(* CODESYS project twinsafe3diagnostics_v0.2.3.library
   Company: Beckhoff Automation LLC - Sample Code
   Version: 0.2.3
   Description: (Sample Code)
   Placeholder: TwinSafe3Diagnostics_v0.2.3
   Author: Jason Erickson
   Title: TwinSafe3Diagnostics_v0.2.3

Project tree, tasks and I/O mapping:
  libraries: Tc2_Drive, * (Beckhoff Automation GmbH); Tc2_EtherCAT, * (Beckhoff Automation GmbH); Tc2_MC2, * (Beckhoff Automation GmbH); Tc2_MC2_Drive, * (Beckhoff Automation GmbH); Tc2_Standard, * (Beckhoff Automation GmbH)
  DUTs/
    ConnectionAndFb_Data/
      FBs/
        data type ST_SAFETY_FB
      Project/
        data type ST_SAFETY_CONNECTION_AX5805
        data type ST_SAFETY_CONNECTION_EK1914
        data type ST_SAFETY_CONNECTION_EL1904
        data type ST_SAFETY_CONNECTION_EL2904
        data type ST_SAFETY_CONNECTION_EP1908
        data type ST_SAFETY_CONNECTION_GROUP
    HardwareData/
      data type ST_AX5805_DIAGNOSTICS
      data type ST_EK1914_DIAGNOSTICS
      data type ST_EL1904_DIAGNOSTICS
      data type ST_EL2904_DIAGNOSTICS
      data type ST_EL69xx_DIAGNOSTICS
      data type ST_EP1908_DIAGNOSTICS
  POUs/
    ConnectionAndFb_Blocks/
      FBs/
        function block FB_InfoAND [ST]
        function block FB_InfoConnectionShutdown [ST]
        function block FB_InfoDecoupler [ST]
        function block FB_InfoEDM [ST]
        function block FB_InfoEStop [ST]
        function block FB_InfoMON [ST]
        function block FB_InfoMuting [ST]
        function block FB_InfoOperationMode [ST]
        function block FB_InfoOR [ST]
        function block FB_InfoRS [ST]
        function block FB_InfoSR [ST]
        function block FB_InfoTOF [ST]
        function block FB_InfoTON [ST]
        function block FB_InfoTwoHand [ST]
      Project/
        function block FB_SafetyConnectionAX5805 [ST]
        function block FB_SafetyConnectionEK1914 [ST]
        function block FB_SafetyConnectionEL1904 [ST]
        function block FB_SafetyConnectionEL2904 [ST]
        function block FB_SafetyConnectionEP1908 [ST]
        function block FB_SafetyConnectionGroup [ST]
    HardwareFBs/
      function block FB_AX5805Diagnostics [ST]
      function block FB_EK1914Diagnostics [ST]
      function block FB_EL1904Diagnostics [ST]
      function block FB_EL2904Diagnostics [ST]
      function block FB_EL69xxDiagnostics [ST]
      function block FB_EP1908Diagnostics [ST]
  Version/
    global variables Global_Version
*)

// DUTs/ConnectionAndFb_Data/FBs/ST_SAFETY_FB
TYPE ST_SAFETY_FB :
STRUCT
(* ***** Structure variables individually linked to the 'Function Block Info Data' of the EL69xx. ***** *)
// State of the TwinSAFE FB.
	usiMapState: USINT;
// Diagnostics of the TwinSAFE FB.
	uiMapDiag: UINT;
END_STRUCT
END_TYPE

// DUTs/ConnectionAndFb_Data/Project/ST_SAFETY_CONNECTION_AX5805
TYPE ST_SAFETY_CONNECTION_AX5805 :
STRUCT
(* ***** Structure linked to the AX5805 'Connection Info Data' of the EL69xx. ***** *)
// State of the AX5805 TwinSAFE connection.
	usiMapState: USINT;
// Diagnostics of the AX5805 TwinSAFE connection.
	usiMapDiag: USINT;
// Connection Input Status signals of the AX5805.
	bInputSignals0: BYTE; // Input status of Channel 1 default motion functions and error.
	bInputSignals1: BYTE; // Input status of Channel 1 USER CONFIGURED motion functions and error.
	bInputSignals2: BYTE; // Input status of Channel 2 default motion functions and error.
	bInputSignals3: BYTE; // Input status of Channel 2 USER CONFIGURED motion functions and error.
// Connection Output Status signals of the AX5805.
	bOutputSignals0: BYTE; // Input status of Channel 1 default motion functions and error.
	bOutputSignals1: BYTE; // Input status of Channel 1 USER CONFIGURED motion functions and error.
	bOutputSignals2: BYTE; // Input status of Channel 2 default motion functions and error.
	bOutputSignals3: BYTE; // Input status of Channel 2 USER CONFIGURED motion functions and error.
END_STRUCT
END_TYPE

// DUTs/ConnectionAndFb_Data/Project/ST_SAFETY_CONNECTION_EK1914
TYPE ST_SAFETY_CONNECTION_EK1914 :
STRUCT
(* ***** Structure linked to the EK1914 'Connection Info Data' of the EL69xx. ***** *)
// State of the EK1914 TwinSAFE connection.
	usiMapState: USINT;
// Diagnostics of the EK1914 TwinSAFE connection.
	usiMapDiag: USINT;
// Input Safe Data Byte 0 of the EK1914.
	bInputSignals: BYTE;
// Output Safe Data Byte 0 of the EK1914.
	bOutputSignals: BYTE;
END_STRUCT
END_TYPE

// DUTs/ConnectionAndFb_Data/Project/ST_SAFETY_CONNECTION_EL1904
TYPE ST_SAFETY_CONNECTION_EL1904 :
STRUCT
(* ***** Structure linked to the EL1904 'Connection Info Data' of the EL69xx. ***** *)
// State of the EL1904 TwinSAFE connection.
	usiMapState: USINT;
// Diagnostics of the EL1904 TwinSAFE connection.
	usiMapDiag: USINT;
// Input Safe Data Byte 0 of the EL1904.
	bInputSignals: BYTE;
END_STRUCT
END_TYPE

// DUTs/ConnectionAndFb_Data/Project/ST_SAFETY_CONNECTION_EL2904
TYPE ST_SAFETY_CONNECTION_EL2904 :
STRUCT
(* ***** Structure linked to the EL2904 'Connection Info Data' of the EL69xx. ***** *)
// State of the EL2904 TwinSAFE connection.
	usiMapState: USINT;
// Diagnostics of the EL2904 TwinSAFE connection.
	usiMapDiag: USINT;
// Output Safe Data Byte 0 of the EL2904.
	bOutputSignals: BYTE;
END_STRUCT
END_TYPE

// DUTs/ConnectionAndFb_Data/Project/ST_SAFETY_CONNECTION_EP1908
TYPE ST_SAFETY_CONNECTION_EP1908 :
STRUCT
(* ***** Structure linked to the EP1908 'Connection Info Data' of the EL69xx. ***** *)
// State of the EP1908 TwinSAFE connection.
	usiMapState: USINT;
// Diagnostics of the EP1908 TwinSAFE connection.
	usiMapDiag: USINT;
// Input Safe Data Byte 0 of the EP1908.
	bInputSignals: BYTE;
END_STRUCT
END_TYPE

// DUTs/ConnectionAndFb_Data/Project/ST_SAFETY_CONNECTION_GROUP
TYPE ST_SAFETY_CONNECTION_GROUP :
STRUCT
(* ***** Structure linked to the 'TwinSAFE Group Info Data' of the EL69xx. ***** *)
// State of the EL2904 TwinSAFE Group.
	usiMapState: USINT;
// Diagnostics of the TwinSAFE Group.
	usiMapDiag: USINT;
END_STRUCT
END_TYPE

// DUTs/HardwareData/ST_AX5805_DIAGNOSTICS
TYPE ST_AX5805_DIAGNOSTICS :
STRUCT
// Serial number of the AX5805.
	dwSerialNumber: DWORD;
// DIP Switch setting of the AX5805.
	wDipSwitch: WORD;
// Hardware Version of the AX5805.
	sHwVersion: STRING(2);
// Software/Firmware Version of the AX5805.
	sFwVersion: STRING(2);
// Micro Controller (MC1) Temperature in DegC of the AX5805.
	wMC1Temp: WORD;
	xMC1_TempHighAlarm: BOOL;
	xMC1_TempLowAlarm: BOOL;
// Micro Controller (MC2) Temperature in DegC of the AX5805.
	wMC2Temp: WORD;
	xMC2_TempHighAlarm: BOOL;
	xMC2_TempLowAlarm: BOOL;
// Micro Controller (MC1) Voltage in mV of the AX5805.
	lrMC1_3300mV: LREAL;
	lrMC1_5000mV: LREAL;
	xMC1_SupplyVoltHighAlarm: BOOL;
	xMC1_SupplyVoltLowAlarm: BOOL;
// Micro Controller (MC2) Voltage (mV) of the AX5805.
	lrMC2_3300mV: LREAL;
	lrMC2_5000mV: LREAL;
	xMC2_SupplyVoltHighAlarm: BOOL;
	xMC2_SupplyVoltLowAlarm: BOOL;
// Configured Safety Option of the AX5000 Drive.
	sSafetyOption: STRING(25);
// Diagnostics outputs of the AX5805.
	sDiagReason: STRING(255);
	sDiagReaction: STRING;
	xDiagnosticAlarm: BOOL;
	iDiagIndex: INT;
// Error outputs of the AX5805.
	sErrorName: STRING;
	sErrorDescription: STRING(255);
	xErrorAlarm: BOOL;
	iErrorIndex: INT;
// Connection State of the AX5805.
	sConnectionState: STRING;
// Error Status of the AX5805.
	xAX5805Error: BOOL;
END_STRUCT
END_TYPE

// DUTs/HardwareData/ST_EK1914_DIAGNOSTICS
TYPE ST_EK1914_DIAGNOSTICS :
STRUCT
// Serial number of the EK1914.
	dwSerialNumber: DWORD;
// DIP Switch setting of the EK1914.
	wDipSwitch: WORD;
// Hardware version of the EK1914.
	sHwVersion: STRING;
// Software/Firmware version of the EK1914.
	sFwVersion: STRING;
// Micro Controller Temperature in DegC of the EK1914.
	wMC1Temp: WORD;
	wMC2Temp: WORD;
// Micro Controller Voltage in mV of the EK1914.
	lrMC1_3300mV: LREAL;
	lrMC2_3300mV: LREAL;
// Sensor Tests Active of the EK1914.
	xSensorTestActive1: BOOL;
	xSensorTestActive2: BOOL;
// Sensor Test Errors of the EK1914.
	xSensorTest1_Error: BOOL;
	xSensorTest2_Error: BOOL;
// Logic Mode of the EK1914 Channels 1 & 2.
	sLogicMode_Ch1Ch2: STRING;
// Standard Output Active/Inactive of the EK1914.
	xStandardOutputActive: BOOL;	
//Test Pulses Active/Inactive of the EK1914.
	xTestPulsesActive: BOOL;
//Output Error Acknowledge Active/Inactive of the EK1914.
	xOutputErrAckActive: BOOL;
// Two-Channel Evaluation Error of the EK1914.
	x2ChanEvalError_Pair1: BOOL;
// Safety Mat Mode Error of the EK1914.
	xSafeMatError_Pair1: BOOL;
// Safety Mat External Supply error of the EK1914.
	xSafeMatExternalSupplyErrorCh1: BOOL;
	xSafeMatExternalSupplyErrorCh2: BOOL;
// Error At The Output of the EK1914 (MC1).
	sOutputErrorDescription_MC1: STRING;
	xCrossCircuitError1_MC1: BOOL;
	xCrossCircuitError2_MC1: BOOL;
	xOverVoltage_MC1: BOOL;
	xUnderVoltage_MC1: BOOL;
	xFieldVoltageError_MC1: BOOL;
	xStartupOutCircuitError_MC1: BOOL;
	xExternalSupply0vError1_MC1: BOOL;
	xExternalSupply24vError1_MC1: BOOL;
	xExternalSupply0vError2_MC1: BOOL;
	xExternalSupply24vError2_MC1: BOOL;
// Error At The Output of the EK1914 (MC2).
	sOutputErrorDescription_MC2: STRING;
	xCrossCircuitError1_MC2: BOOL;
	xCrossCircuitError2_MC2: BOOL;
	xOverVoltage_MC2: BOOL;
	xUnderVoltage_MC2: BOOL;
	xFieldVoltageError_MC2: BOOL;
	xStartupOutCircuitError_MC2: BOOL;
	xExternalSupply0vError1_MC2: BOOL;
	xExternalSupply24vError1_MC2: BOOL;
	xExternalSupply0vError2_MC2: BOOL;
	xExternalSupply24vError2_MC2: BOOL;
// Connection State of the EK1914.
	sConnectionState: STRING;
// Error Status of the EK1914.
	xEK1914Error: BOOL;
END_STRUCT
END_TYPE

// DUTs/HardwareData/ST_EL1904_DIAGNOSTICS
TYPE ST_EL1904_DIAGNOSTICS :
STRUCT
// Serial number of the EL1904.
	dwSerialNumber: DWORD;
// DIP Switch setting of the EL1904.
	wDipSwitch: WORD;
// Hardware version of the EL1904.
	sHwVersion: STRING;
// Software/Firmware version of the EL1904.
	sFwVersion: STRING;
// Micro Controller Temperature in DegC of the EL1904.
	wMC1Temp: WORD;
	wMC2Temp: WORD;
// Micro Controller Voltage in mV of the EL1904.
	lrMC1_3300mV: LREAL;
	lrMC2_3300mV: LREAL;
// Operating Mode of the EL1904.
	sOpMode: STRING;
// Sensor Tests Active of the EL1904.
	xSensorTestActive1: BOOL;
	xSensorTestActive2: BOOL;
	xSensorTestActive3: BOOL;
	xSensorTestActive4: BOOL;
// Sensor Test Errors of the EL1904.
	xSensorTest1_Error: BOOL;
	xSensorTest2_Error: BOOL;
	xSensorTest3_Error: BOOL;
	xSensorTest4_Error: BOOL;
// Logic Mode of the EL1904 Channels 1 & 2.
	sLogicMode_Ch1Ch2: STRING;
// Logic Mode of the EL1904 Channels 3 & 4.
	sLogicMode_Ch3Ch4: STRING;
// Two-Channel Evaluation Error of the EL1904.
	x2ChanEvalError_Pair1: BOOL;
	x2ChanEvalError_Pair2: BOOL;
// Safety Mat Mode Error of the EL1904.
	xSafeMatError_Pair1: BOOL;
	xSafeMatError_Pair2: BOOL;
// Safety Mat External Supply error of the EL1904.
	xSafeMatExternalSupplyErrorCh1: BOOL;
	xSafeMatExternalSupplyErrorCh2: BOOL;
	xSafeMatExternalSupplyErrorCh3: BOOL;
	xSafeMatExternalSupplyErrorCh4: BOOL;
// Connection State of the EL1904.
	sConnectionState: STRING;
// Error Status of the EL1904.
	xEL1904Error: BOOL;
END_STRUCT
END_TYPE

// DUTs/HardwareData/ST_EL2904_DIAGNOSTICS
TYPE ST_EL2904_DIAGNOSTICS :
STRUCT
// Serial number of the EL2904.
	dwSerialNumber: DWORD;
// DIP Switch setting of the EL2904.
	wDipSwitch: WORD;
// Hardware version of the EL2904.
	sHwVersion: STRING;
// Software/Firmware version of the EL2904.
	sFwVersion: STRING;
// Micro Controller Temperature in DegC of the EL2904.
	wMC1Temp: WORD;
	wMC2Temp: WORD;
// Micro Controller Voltage in mV of the EL2904.
	lrMC1_3300mV: LREAL;
	lrMC2_3300mV: LREAL;
// Standard Output Active/Inactive of the EL2904.
	xStandardOutputActive: BOOL;	
// Current Measurement Active of the EL2904.
	xCurrentMeasureActive: BOOL;
//Test Pulses Active/Inactive of the EL2904.
	xTestPulsesActive: BOOL;
//Output Error Acknowledge Active/Inactive of the EL2904.
	xOutputErrAckActive: BOOL;
// Error At The Output of the EL2904.
	xExternalSupplyOrCrossCircuitError1: BOOL;
	xExternalSupplyOrCrossCircuitError2: BOOL;
	xExternalSupplyOrCrossCircuitError3: BOOL;
	xExternalSupplyOrCrossCircuitError4: BOOL;
	xLoadError1: BOOL;
	xLoadError2: BOOL;
	xLoadError3: BOOL;
	xLoadError4: BOOL;
//Power Rail Supply Error of the EL2904
	xPowerRailSupplyVoltHighError: BOOL;
	xPowerRailSupplyVoltLowError: BOOL;
// Internal Chip Temperature Error of the EL2904.
	xOverTempMC1: BOOL;
	xOverTempMC2: BOOL;
	xOverTempOutputBoard: BOOL;
	xUnderTempMC1: BOOL;
	xUnderTempMC2: BOOL;
	xUnderTempOutputBoard: BOOL;
	xTempDiffOutputBoard: BOOL;
	xTempDiff_MC1MC2: BOOL;
// Connection State of the EL2904.
	sConnectionState: STRING;
// Error Status of the EL2904.
	xEL2904Error: BOOL;
END_STRUCT
END_TYPE

// DUTs/HardwareData/ST_EL69xx_DIAGNOSTICS
TYPE ST_EL69xx_DIAGNOSTICS :
STRUCT
// Serial number of the EL69xx.
	dwSerialNumber: DWORD;
// DIP Switch setting of the EL69xx.
	wDipSwitch: WORD;
// Hardware version of the EL69xx.
	sHwVersion: STRING;
// Software/Firmware version of the EL69xx.
	sFwVersion: STRING;
// Micro Controller Temperature in DegC of the EL69xx.
	wMC1Temp: WORD;
	wMC2Temp: WORD;
// Micro Controller voltage in mV of the EL69xx.
	lrMC1_3300mV: LREAL;
	lrMC2_3300mV: LREAL;
// Temperature and Voltage Errors of the EL69xx.
	xMaxTempError: BOOL;
	xMinTempError: BOOL;
	xTempDiffError: BOOL;
	xMaxVccMC1: BOOL;
	xMaxVccMC2: BOOL;
	xMinVccMC1: BOOL;
	xMinVccMC2: BOOL;
// Number Of Connections Configured in the EL69xx.
	bNumOfConnections: BYTE;
// Number of Safety Groups Configured in the EL69xx.
	bNumOfSafetyGroups: BYTE;
//Number of Safety Function Blocks Configured in the EL69xx.
	bNumOfSafetyBlocks: BYTE;
// Error Status of the EL69xx.
	xEL69xxError: BOOL;
END_STRUCT
END_TYPE

// DUTs/HardwareData/ST_EP1908_DIAGNOSTICS
TYPE ST_EP1908_DIAGNOSTICS :
STRUCT
// Serial number of the EP1908.
	dwSerialNumber: DWORD;
// DIP Switch setting of the EP1908.
	wDipSwitch: WORD;
// Hardware version of the EP1908.
	sHwVersion: STRING;
// Software/Firmware version of the EP1908.
	sFwVersion: STRING;
// Micro Controller Temperature in DegC of the EP1908.
	wMC1Temp: WORD;
	wMC2Temp: WORD;
// Micro Controller Voltage in mV of the EP1908.
	lrMC1_3300mV: LREAL;
	lrMC2_3300mV: LREAL;
// Operating Mode of the EP1908.
	sOpMode: STRING;
// Sensor Tests Active of the EP1908.
	xSensorTestActive1: BOOL;
	xSensorTestActive2: BOOL;
	xSensorTestActive3: BOOL;
	xSensorTestActive4: BOOL;
	xSensorTestActive5: BOOL;
	xSensorTestActive6: BOOL;
	xSensorTestActive7: BOOL;
	xSensorTestActive8: BOOL;
// Sensor Test Errors of the EP1908.
	xSensorTest1_Error: BOOL;
	xSensorTest2_Error: BOOL;
	xSensorTest3_Error: BOOL;
	xSensorTest4_Error: BOOL;
	xSensorTest5_Error: BOOL;
	xSensorTest6_Error: BOOL;
	xSensorTest7_Error: BOOL;
	xSensorTest8_Error: BOOL;
// Logic Mode 1 & 2 of the EP1908.
	sLogicMode_Ch1Ch2: STRING;
// Logic Mode 3 & 4 of the EP1908.
	sLogicMode_Ch3Ch4: STRING;
// Logic Mode 5 & 6 of the EP1908.
	sLogicMode_Ch5Ch6: STRING;
// Logic Mode 7 & 8 of the EP1908.
	sLogicMode_Ch7Ch8: STRING;
// Velocity/Frequency Limits of the EP1908.
	iEP1908_VelocityLimitCh1: INT;
	iEP1908_VelocityLimitCh2: INT;
	iEP1908_VelocityLimitCh3: INT;
	iEP1908_VelocityLimitCh4: INT;
	iEP1908_VelocityLimitCh5: INT;
	iEP1908_VelocityLimitCh6: INT;
	iEP1908_VelocityLimitCh7: INT;
	iEP1908_VelocityLimitCh8: INT;
// Actual Velocity/Frequencies of the EP1908.
 	iEP1908_ActVeloctiyCh1: INT;
 	iEP1908_ActVeloctiyCh2: INT;
 	iEP1908_ActVeloctiyCh3: INT;
 	iEP1908_ActVeloctiyCh4: INT;
 	iEP1908_ActVeloctiyCh5: INT;
 	iEP1908_ActVeloctiyCh6: INT;
 	iEP1908_ActVeloctiyCh7: INT;
 	iEP1908_ActVeloctiyCh8: INT;
// Max Velocitys/Frequencies of the EP1908.
	iEP1908_MaxVeloctiyCh1: INT;
	iEP1908_MaxVeloctiyCh2: INT;
	iEP1908_MaxVeloctiyCh3: INT;
	iEP1908_MaxVeloctiyCh4: INT;
	iEP1908_MaxVeloctiyCh5: INT;
	iEP1908_MaxVeloctiyCh6: INT;
	iEP1908_MaxVeloctiyCh7: INT;
	iEP1908_MaxVeloctiyCh8: INT;
// Two-Channel Evaluation Error of the EP1908.
	x2ChanEvalError_Pair1: BOOL;
	x2ChanEvalError_Pair2: BOOL;
	x2ChanEvalError_Pair3: BOOL;
	x2ChanEvalError_Pair4: BOOL;
// Safety Mat Mode Error of the EP1908.
	xSafeMatError_Pair1: BOOL;
	xSafeMatError_Pair2: BOOL;
	xSafeMatError_Pair3: BOOL;
	xSafeMatError_Pair4: BOOL;
// Safety Mat External Supply error of the EP1908.
	xSafeMatExternalSupplyErrorCh1: BOOL;
	xSafeMatExternalSupplyErrorCh2: BOOL;
	xSafeMatExternalSupplyErrorCh3: BOOL;
	xSafeMatExternalSupplyErrorCh4: BOOL;
	xSafeMatExternalSupplyErrorCh5: BOOL;
	xSafeMatExternalSupplyErrorCh6: BOOL;
	xSafeMatExternalSupplyErrorCh7: BOOL;
	xSafeMatExternalSupplyErrorCh8: BOOL;
// Speed Monitoring Error: Overspeed of the EP1908. 
// (Overspeed was detected at the input).
	xSpeedMonitorErrorCh1: BOOL;
	xSpeedMonitorErrorCh2: BOOL;
	xSpeedMonitorErrorCh3: BOOL;
	xSpeedMonitorErrorCh4: BOOL;
	xSpeedMonitorErrorCh5: BOOL;
	xSpeedMonitorErrorCh6: BOOL;
	xSpeedMonitorErrorCh7: BOOL;
	xSpeedMonitorErrorCh8: BOOL;
// Two Channel Sync Velocity Control Error of the EP1908. 
// (Both inputs of an input pair were read with inactive State).
	x2ChSyncVelocityErrorPair1: BOOL;
	x2ChSyncVelocityErrorPair2: BOOL;
	x2ChSyncVelocityErrorPair3: BOOL;
	x2ChSyncVelocityErrorPair4: BOOL;
// Two Channel Sync Velocity AND Two Channel Encoder Velocity Error of the EP1908.
// (Different speeds were identified for the two inputs of an input pair).
	x2ChSyncVeloAnd2ChEncVeloErrorPair1: BOOL;
	x2ChSyncVeloAnd2ChEncVeloErrorPair2: BOOL;
	x2ChSyncVeloAnd2ChEncVeloErrorPair3: BOOL;
	x2ChSyncVeloAnd2ChEncVeloErrorPair4: BOOL;
// Connection State of the EP1908.
	sConnectionState: STRING;
// Error Status of the EP1908.
	xEP1908Error: BOOL;
END_STRUCT
END_TYPE

// Version/Global_Version
// This function has been automatically generated from the project information.
VAR_GLOBAL CONSTANT
	{attribute 'const_non_replaced'}
	{attribute 'linkalways'}
	stLibVersion_TwinSafe3Diagnostics_v0_2_3 : ST_LibVersion := (iMajor := 0, iMinor := 2, iBuild := 3, iRevision := 0, sVersion := '0.2.3');
END_VAR

// POUs/ConnectionAndFb_Blocks/FBs/FB_InfoAND
(*=====================================================================
Beckhoff Automation LLC
Copyright 2015 All Rights Reserved
=======================================================================
Description: 
This Program has been supplied by Beckhoff Automation As-Is and is intended only as an example implementation. 
Functionality is not guaranteed. 
This Function Block reads status and error information known at time of creation of the TwinSAFE 'safeAnd' 
function block.
---------------------------------------------------------------------------------------------------------------
History:
Date		Version			Author							Comment
---------------------------------------------------------------------------------------------------------------
07.08.15	0.10		Jason Erickson				Initial Library Creation.
07.20.15	0.11		Jason Ericskon				Added CoE Read for TwinSAFE Connection State.
08.28.15	0.20		Jason Erickson				Code optimization to eliminate timed data reads.
09.18.15	0.2.1		Jason Erickson				Added new error codes 0x6000 - 0x6002 and Connection Status
														to the AX5805.
*)
FUNCTION_BLOCK FB_InfoAND
VAR_INPUT
(* ***** Structure variables individually linked to the 'Function Block Info Data' of the EL69xx. ***** *)
	i_stInfoData: ST_SAFETY_FB ;
END_VAR
VAR_OUTPUT
// State of the TwinSAFE FB.
	q_sState: STRING ;
END_VAR

// Evaluate safeAnd FB State.
IF i_stInfoData.usiMapState = 0 THEN
	q_sState := 'Undefined' ;
	ELSIF i_stInfoData.usiMapState 	= 	1 THEN
		q_sState := 'RUN' ;
	ELSIF i_stInfoData.usiMapState = 2 THEN
		q_sState := 'STOP' ;
	ELSIF i_stInfoData.usiMapState = 3 THEN
		q_sState := 'SAFE' ;
	ELSE
		q_sState := 'Unknown' ;
END_IF

// THE 'safeAnd' FB HAS NO DIAGNISTIC BYTE TO DECODE!

END_FUNCTION_BLOCK

// POUs/ConnectionAndFb_Blocks/FBs/FB_InfoConnectionShutdown
(*=====================================================================
Beckhoff Automation LLC
Copyright 2015 All Rights Reserved
=======================================================================
Description: 
This Program has been supplied by Beckhoff Automation As-Is and is intended only as an example implementation. 
Functionality is not guaranteed. 
This Function Block reads status and error information known at time of creation of the TwinSAFE 'safeConnShutdown' 
function block.
---------------------------------------------------------------------------------------------------------------
History:
Date		Version			Author							Comment
---------------------------------------------------------------------------------------------------------------
07.08.15	0.10		Jason Erickson				Initial Library Creation.
07.20.15	0.11		Jason Ericskon				Added CoE Read for TwinSAFE Connection State.
08.28.15	0.20		Jason Erickson				Code optimization to eliminate timed data reads.
09.18.15	0.2.1		Jason Erickson				Added new error codes 0x6000 - 0x6002 and Connection Status
														to the AX5805.
*)
FUNCTION_BLOCK FB_InfoConnectionShutdown
VAR_INPUT
(* ***** Structure variables individually linked to the 'Function Block Info Data' of the EL69xx. ***** *)
	i_stInfoData: ST_SAFETY_FB ;
END_VAR
VAR_OUTPUT
// State of the TwinSAFE FB.
	q_sState: STRING ;
// Diagnostics of the TwinSAFE FB.
	q_sDiag: STRING ;
END_VAR

// Evaluate safeConnShutdown FB State.
IF i_stInfoData.usiMapState = 0 THEN
	q_sState := 'Undefined' ;
	ELSIF i_stInfoData.usiMapState = 2 THEN
		q_sState := 'STOP' ;
	ELSIF i_stInfoData.usiMapState 	= 	3 THEN
		q_sState := 'SAFE' ;
	ELSIF i_stInfoData.usiMapState = 4 THEN
		q_sState := 'Error' ;
	ELSIF i_stInfoData.usiMapState = 5 THEN
		q_sState := 'Reset' ;
	ELSIF i_stInfoData.usiMapState = 10 THEN
		q_sState := 'Active' ;
	ELSIF i_stInfoData.usiMapState = 11 THEN
		q_sState := 'Deactive' ;
	ELSE
		q_sState := 'Unknown' ;
END_IF

// Evaluate safeConnShutdown FB Diagnostics.
IF i_stInfoData.uiMapDiag = 0 THEN
	q_sDiag := 'No Error' ;
	ELSIF  i_stInfoData.uiMapDiag = 1 THEN
		q_sDiag := 'Discrepancy Error Input Group1' ;
	ELSE
		q_sDiag := 'Unknown' ;
END_IF

END_FUNCTION_BLOCK

// POUs/ConnectionAndFb_Blocks/FBs/FB_InfoDecoupler
(*=====================================================================
Beckhoff Automation LLC
Copyright 2015 All Rights Reserved
=======================================================================
Description: 
This Program has been supplied by Beckhoff Automation As-Is and is intended only as an example implementation. 
Functionality is not guaranteed. 
This Function Block reads status and error information known at time of creation of the TwinSAFE 'safeDecouple' 
function block.
---------------------------------------------------------------------------------------------------------------
History:
Date		Version			Author							Comment
---------------------------------------------------------------------------------------------------------------
07.08.15	0.10		Jason Erickson				Initial Library Creation.
07.20.15	0.11		Jason Ericskon				Added CoE Read for TwinSAFE Connection State.
08.28.15	0.20		Jason Erickson				Code optimization to eliminate timed data reads.
09.18.15	0.2.1		Jason Erickson				Added new error codes 0x6000 - 0x6002 and Connection Status
														to the AX5805.
*)
FUNCTION_BLOCK FB_InfoDecoupler
VAR_INPUT
(* ***** Structure variables individually linked to the 'Function Block Info Data' of the EL69xx. ***** *)
	i_stInfoData: ST_SAFETY_FB ;
END_VAR
VAR_OUTPUT
// State of the TwinSAFE FB.
	q_sState: STRING ;
END_VAR

// Evaluate safeDecouple FB State.
IF i_stInfoData.usiMapState = 0 THEN
	q_sState := 'Undefined' ;
	ELSIF i_stInfoData.usiMapState = 1 THEN
		q_sState := 'RUN' ;
	ELSIF i_stInfoData.usiMapState = 2 THEN
		q_sState := 'STOP' ;
	ELSE
		q_sState := 'Unknown' ;
END_IF

// THE 'DECOUPLE FB' HAS NO DIAGNOSTIC BYTE TO DECODE!

END_FUNCTION_BLOCK

// POUs/ConnectionAndFb_Blocks/FBs/FB_InfoEDM
(*=====================================================================
Beckhoff Automation LLC
Copyright 2015 All Rights Reserved
=======================================================================
Description: 
This Program has been supplied by Beckhoff Automation As-Is and is intended only as an example implementation. 
Functionality is not guaranteed. 
This Function Block reads status and error information known at time of creation of the TwinSAFE 'safeEdm' 
function block.
---------------------------------------------------------------------------------------------------------------
History:
Date		Version			Author							Comment
---------------------------------------------------------------------------------------------------------------
07.08.15	0.10		Jason Erickson				Initial Library Creation.
07.20.15	0.11		Jason Ericskon				Added CoE Read for TwinSAFE Connection State.
08.28.15	0.20		Jason Erickson				Code optimization to eliminate timed data reads.
09.18.15	0.2.1		Jason Erickson				Added new error codes 0x6000 - 0x6002 and Connection Status
														to the AX5805.
*)
FUNCTION_BLOCK FB_InfoEDM
VAR_INPUT
(* ***** Structure variables individually linked to the 'Function Block Info Data' of the EL69xx. ***** *)
	i_stInfoData: ST_SAFETY_FB ;
END_VAR
VAR_OUTPUT
// State of the TwinSAFE FB.
	q_sState: STRING ;
// Diagnostics of the TwinSAFE FB.
	q_sDiag: STRING ;
END_VAR

// Evaluate safeEdm FB State.
IF i_stInfoData.usiMapState = 0 THEN
				q_sState := 'Undefined' ;
	ELSIF i_stInfoData.usiMapState = 2 THEN
				q_sState := 'STOP' ;
	ELSIF i_stInfoData.usiMapState = 4 THEN
				q_sState := 'ERROR' ;
	ELSIF i_stInfoData.usiMapState 	= 	5 THEN
				q_sState := 'RESET' ;
	ELSIF i_stInfoData.usiMapState = 14 THEN
				q_sState := 'Monitor-OFF' ;
	ELSIF i_stInfoData.usiMapState = 15 THEN
				q_sState := 'Monitor-ON' ;
	ELSE
				q_sState := 'Unknown' ;
END_IF

// Evaluate safeEdm FB Diagnostics
IF i_stInfoData.uiMapDiag = 0 THEN
				q_sDiag := 'No Error' ;
ELSIF  i_stInfoData.uiMapDiag = 1 THEN
				q_sDiag	:= 'Switch-OFF Timer Elapsed' ;
ELSIF  i_stInfoData.uiMapDiag = 2 THEN
				q_sDiag := 'Switch-ON Timer Elapsed' ;
ELSE
				q_sDiag := 'Unknown' ;
END_IF

END_FUNCTION_BLOCK

// POUs/ConnectionAndFb_Blocks/FBs/FB_InfoEStop
(*=====================================================================
Beckhoff Automation LLC
Copyright 2015 All Rights Reserved
=======================================================================
Description: 
This Program has been supplied by Beckhoff Automation As-Is and is intended only as an example implementation. 
Functionality is not guaranteed. 
This Function Block reads status and error information known at time of creation of the TwinSAFE 'safeEstop' 
function block.
---------------------------------------------------------------------------------------------------------------
History:
Date		Version			Author							Comment
---------------------------------------------------------------------------------------------------------------
07.08.15	0.10		Jason Erickson				Initial Library Creation.
07.20.15	0.11		Jason Ericskon				Added CoE Read for TwinSAFE Connection State.
08.28.15	0.20		Jason Erickson				Code optimization to eliminate timed data reads.
09.18.15	0.2.1		Jason Erickson				Added new error codes 0x6000 - 0x6002 and Connection Status
														to the AX5805.
*)
FUNCTION_BLOCK FB_InfoEStop
VAR_INPUT
(* ***** Structure variables individually linked to the 'Function Block Info Data' of the EL69xx. ***** *)
	i_stInfoData: ST_SAFETY_FB ;
END_VAR
VAR_OUTPUT
// State of the TwinSAFE FB.
	q_sState: STRING ;
// Diagnostics of the TwinSAFE FB.
	q_sDiag: STRING ;
END_VAR

// Evaluate state of the TwinSAFE 'ESTOP' FB.
IF i_stInfoData.usiMapState = 0 THEN
	q_sState := 'Undefined' ;
	ELSIF i_stInfoData.usiMapState = 1 THEN
		q_sState := 'RUN' ;
	ELSIF i_stInfoData.usiMapState = 2 THEN
		q_sState := 'STOP' ;
	ELSIF i_stInfoData.usiMapState = 3 THEN
		q_sState := 'SAFE' ;
	ELSIF i_stInfoData.usiMapState = 4 THEN
		q_sState := 'ERROR' ;
	ELSIF i_stInfoData.usiMapState = 5 THEN
		q_sState := 'RESET' ;
	ELSIF i_stInfoData.usiMapState = 6 THEN
		q_sState := 'START' ;
	ELSIF i_stInfoData.usiMapState = 8 THEN
		q_sState := 'DELAYOUT' ;
	ELSE
		q_sState := 'Unknown' ;
END_IF

// Evaluate diagnostics of the TwinSAFE 'ESTOP' FB.
IF i_stInfoData.uiMapDiag = 0 THEN
	q_sDiag := 'No Error' ;
	ELSIF i_stInfoData.uiMapDiag = 1 THEN
		q_sDiag := 'Discrepancy Error Input Group 1' ;
	ELSIF i_stInfoData.uiMapDiag = 2 THEN
		q_sDiag := 'Discrepancy Error Input Group 2' ;
	ELSIF i_stInfoData.uiMapDiag = 4 THEN
		q_sDiag := 'Discrepancy Error Input Group 3' ;
	ELSIF i_stInfoData.uiMapDiag = 8 THEN
		q_sDiag := 'Discrepancy Error Input Group 4' ;
	ELSIF i_stInfoData.uiMapDiag = 16 THEN
		q_sDiag := 'EDM 1 Monitoring Error' ;	
	ELSIF i_stInfoData.uiMapDiag = 32 THEN
		q_sDiag :=  	'EDM 2 Monitoring Error' ;	
	ELSE
		q_sDiag := 'Unknown' ;
END_IF

END_FUNCTION_BLOCK

// POUs/ConnectionAndFb_Blocks/FBs/FB_InfoMON
(*=====================================================================
Beckhoff Automation LLC
Copyright 2015 All Rights Reserved
=======================================================================
Description: 
This Program has been supplied by Beckhoff Automation As-Is and is intended only as an example implementation. 
Functionality is not guaranteed. 
This Function Block reads status and error information known at time of creation of the TwinSAFE 'safeMon' 
function block.
---------------------------------------------------------------------------------------------------------------
History:
Date		Version			Author							Comment
---------------------------------------------------------------------------------------------------------------
07.08.15	0.10		Jason Erickson				Initial Library Creation.
07.20.15	0.11		Jason Ericskon				Added CoE Read for TwinSAFE Connection State.
08.28.15	0.20		Jason Erickson				Code optimization to eliminate timed data reads.
09.18.15	0.2.1		Jason Erickson				Added new error codes 0x6000 - 0x6002 and Connection Status
														to the AX5805.
*)
FUNCTION_BLOCK FB_InfoMON
VAR_INPUT
(* ***** Structure variables individually linked to the 'Function Block Info Data' of the EL69xx. ***** *)
	i_stInfoData: ST_SAFETY_FB ;
END_VAR
VAR_OUTPUT
// State of the TwinSAFE FB.
	q_sState: STRING ;
// Diagnostics of the TwinSAFE FB.
	q_sDiag: STRING ;
END_VAR

// Evaluate state of the TwinSAFE 'safeMon' FB.
IF i_stInfoData.usiMapState = 0 THEN
	q_sState := 'Undefined' ;
	ELSIF i_stInfoData.usiMapState = 1 THEN
		q_sState := 'RUN' ;
	ELSIF i_stInfoData.usiMapState = 2 THEN
		q_sState := 'STOP' ;
	ELSIF i_stInfoData.usiMapState = 3 THEN
		q_sState := 'SAFE' ;
	ELSIF i_stInfoData.usiMapState = 4 THEN
		q_sState := 'ERROR' ;
	ELSIF i_stInfoData.usiMapState = 5 THEN
		q_sState := 'RESET' ;
	ELSIF i_stInfoData.usiMapState = 6 THEN
		q_sState := 'START' ;
	ELSIF i_stInfoData.usiMapState = 7 THEN
		q_sState := 'Error Delay' ;
	ELSIF i_stInfoData.usiMapState = 8 THEN
		q_sState := 	'DelayOut' ;
	ELSIF i_stInfoData.usiMapState = 9 THEN
		q_sState := 'Function Test' ;
	ELSE
		q_sState := 'Unknown' ;
END_IF

// Evaluate diagnostics of the TwinSAFE 'safeMon' FB.
IF i_stInfoData.uiMapDiag = 0 THEN
	q_sDiag := 'No Error' ;
	ELSIF  i_stInfoData.uiMapDiag = 1 THEN
		q_sDiag := 'Discrepancy Error of Input Group 1' ;
	ELSIF  i_stInfoData.uiMapDiag = 2 THEN
		q_sDiag := 'Discrepancy Error of Input Group 2' ;
	ELSIF  i_stInfoData.uiMapDiag = 4 THEN
		q_sDiag := 'Discrepancy Error of the Secure Inputs' ;
	ELSIF  i_stInfoData.uiMapDiag = 16 THEN
		q_sDiag := 'EDM 1 Monitoring Error' ;
	ELSIF  i_stInfoData.uiMapDiag = 32 THEN
		q_sDiag := 'EDM 2 Monitoring Error' ;
	ELSE
		q_sDiag := 'Unknown' ;
END_IF

END_FUNCTION_BLOCK

// POUs/ConnectionAndFb_Blocks/FBs/FB_InfoMuting
(*=====================================================================
Beckhoff Automation LLC
Copyright 2015 All Rights Reserved
=======================================================================
Description: 
This Program has been supplied by Beckhoff Automation As-Is and is intended only as an example implementation. 
Functionality is not guaranteed. 
This Function Block reads status and error information known at time of creation of the TwinSAFE 'safeMuting' 
function block.
---------------------------------------------------------------------------------------------------------------
History:
Date		Version			Author							Comment
---------------------------------------------------------------------------------------------------------------
07.08.15	0.10		Jason Erickson				Initial Library Creation.
07.20.15	0.11		Jason Ericskon				Added CoE Read for TwinSAFE Connection State.
08.28.15	0.20		Jason Erickson				Code optimization to eliminate timed data reads.
09.18.15	0.2.1		Jason Erickson				Added new error codes 0x6000 - 0x6002 and Connection Status
														to the AX5805.
*)
FUNCTION_BLOCK FB_InfoMuting
VAR_INPUT
(* ***** Structure variables individually linked to the 'Function Block Info Data' of the EL69xx. ***** *)
	i_stInfoData: ST_SAFETY_FB ;
END_VAR
VAR_OUTPUT
// State of the TwinSAFE FB.
	q_sState: STRING ;
// Diagnostics of the TwinSAFE FB.
	q_sDiag: STRING ;
END_VAR

// Evaluate state of the TwinSAFE 'safeMuting' FB.
IF i_stInfoData.usiMapState = 0 THEN
	q_sState := 'Undefined' ;
	ELSIF i_stInfoData.usiMapState = 1 THEN
		q_sState := 'RUN' ;
	ELSIF i_stInfoData.usiMapState = 2 THEN
		q_sState := 'STOP' ;
	ELSIF i_stInfoData.usiMapState = 3 THEN
		q_sState := 'SAFE' ;
	ELSIF i_stInfoData.usiMapState = 4 THEN
		q_sState := 'ERROR' ;
	ELSIF i_stInfoData.usiMapState = 5 THEN
		q_sState := 'RESET' ;
	ELSIF i_stInfoData.usiMapState = 8 THEN
		q_sState := 'DelayOut' ;
	ELSIF i_stInfoData.usiMapState = 9 THEN
		q_sState := 'Muting 1' ;
	ELSIF i_stInfoData.usiMapState = 10 THEN
		q_sState := 'Muting 2' ;
	ELSIF i_stInfoData.usiMapState = 11 THEN
		q_sState := 'Muting 3' ;
	ELSIF i_stInfoData.usiMapState = 12 THEN
		q_sState := 'Muting 4' ;
	ELSIF i_stInfoData.usiMapState = 13 THEN
		q_sState := 'Muting 5' ;
	ELSIF i_stInfoData.usiMapState = 14 THEN
		q_sState := 'Muting 6' ;
	ELSIF i_stInfoData.usiMapState = 15 THEN
		q_sState := 'Muting 7' ;
	ELSIF i_stInfoData.usiMapState = 16 THEN
		q_sState := 'Muting 8' ;
	ELSIF i_stInfoData.usiMapState = 17 THEN
		q_sState := 'Muting 9' ;
	ELSE
		q_sState := 'Unknown' ;
END_IF

// Evaluate diagnostics of the TwinSAFE 'safeMuting' FB.
IF i_stInfoData.uiMapDiag = 0 THEN
	q_sDiag := 'No Error' ;
	ELSIF  i_stInfoData.uiMapDiag = 1 THEN
		q_sDiag := 'Discrepancy Error In Muting Input Group 1' ;
	ELSIF  i_stInfoData.uiMapDiag = 2 THEN
		q_sDiag := 'Discrepancy Error In OSSD Input Group' ;
	ELSIF  i_stInfoData.uiMapDiag = 4 THEN
		q_sDiag := 'Discrepancy Error In Muting Input Group 2' ;
	ELSIF  i_stInfoData.uiMapDiag = 16 THEN
		q_sDiag := 'EDM 1 Monitoring Error' ;
	ELSIF  i_stInfoData.uiMapDiag = 32 THEN
		q_sDiag := 'EDM 2 Monitoring Error' ;
	ELSIF  i_stInfoData.uiMapDiag = 64 THEN
		q_sDiag := 'Muting Sequence Was Violated' ;
	ELSIF  i_stInfoData.uiMapDiag = 128 THEN
		q_sDiag := 'Maximum Muting Time Was Exceeded' ;
	ELSE
		q_sDiag := 'Unknown' ;
END_IF

END_FUNCTION_BLOCK

// POUs/ConnectionAndFb_Blocks/FBs/FB_InfoOperationMode
(*=====================================================================
Beckhoff Automation LLC
Copyright 2015 All Rights Reserved
=======================================================================
Description: 
This Program has been supplied by Beckhoff Automation As-Is and is intended only as an example implementation. 
Functionality is not guaranteed.  
This Function Block reads status and error information known at time of creation of the TwinSAFE 'safeOpmode' 
function block.
---------------------------------------------------------------------------------------------------------------
History:
Date		Version			Author							Comment
---------------------------------------------------------------------------------------------------------------
07.08.15	0.10		Jason Erickson				Initial Library Creation.
07.20.15	0.11		Jason Ericskon				Added CoE Read for TwinSAFE Connection State.
08.28.15	0.20		Jason Erickson				Code optimization to eliminate timed data reads.
09.18.15	0.2.1		Jason Erickson				Added new error codes 0x6000 - 0x6002 and Connection Status
														to the AX5805.
*)
FUNCTION_BLOCK FB_InfoOperationMode
VAR_INPUT
(* ***** Structure variables individually linked to the 'Function Block Info Data' of the EL69xx. ***** *)
	i_stInfoData: ST_SAFETY_FB ;
END_VAR
VAR_OUTPUT
// State of the TwinSAFE FB.
	q_sState: STRING ;
// Diagnostics of the TwinSAFE FB.
	q_sDiag: STRING ;
END_VAR

// Evaluate safeOpmode FB State.
IF i_stInfoData.usiMapState = 0 THEN
	q_sState := 'Undefined' ;
	ELSIF i_stInfoData.usiMapState = 1 THEN
		q_sState := 'RUN' ;
	ELSIF i_stInfoData.usiMapState = 2 THEN
		q_sState := 'STOP' ;
	ELSIF i_stInfoData.usiMapState = 3 THEN
		q_sState := 'SAFE' ;
	ELSIF i_stInfoData.usiMapState = 4 THEN
		q_sState := 'ERROR' ;
	ELSIF i_stInfoData.usiMapState = 5 THEN
		q_sState := 'RESET' ;
	ELSIF i_stInfoData.usiMapState = 6 THEN
		q_sState := 'START' ;
	ELSE
		q_sState := 'Unknown' ;
END_IF

// Evaluate safeOpmode FB Diagnostics
IF i_stInfoData.uiMapDiag=0 THEN
	q_sDiag:='No Error' ;
	ELSIF  i_stInfoData.uiMapDiag=1 THEN
		q_sDiag:='Discrepancy Monitoring Error' ;
	ELSE
		q_sDiag:='Unknown' ;
END_IF

END_FUNCTION_BLOCK

// POUs/ConnectionAndFb_Blocks/FBs/FB_InfoOR
(*=====================================================================
Beckhoff Automation LLC
Copyright 2015 All Rights Reserved
=======================================================================
Description: 
This Program has been supplied by Beckhoff Automation As-Is and is intended only as an example implementation. 
Functionality is not guaranteed. 
This Function Block reads status and error information known at time of creation of the TwinSAFE 'safeOr' 
function block.
---------------------------------------------------------------------------------------------------------------
History:
Date		Version			Author							Comment
---------------------------------------------------------------------------------------------------------------
07.08.15	0.10		Jason Erickson				Initial Library Creation.
07.20.15	0.11		Jason Ericskon				Added CoE Read for TwinSAFE Connection State.
08.28.15	0.20		Jason Erickson				Code optimization to eliminate timed data reads.
09.18.15	0.2.1		Jason Erickson				Added new error codes 0x6000 - 0x6002 and Connection Status
														to the AX5805.
*)
FUNCTION_BLOCK FB_InfoOR
VAR_INPUT
(* ***** Structure variables individually linked to the 'Function Block Info Data' of the EL69xx. ***** *)
	i_stInfoData: ST_SAFETY_FB ;
END_VAR
VAR_OUTPUT
// State of the TwinSAFE FB.
	q_sState: STRING ;
END_VAR

// Evaluate state of the TwinSAFE 'safeOr' FB.
IF i_stInfoData.usiMapState = 0 THEN
	q_sState := 'Undefined' ;
	ELSIF i_stInfoData.usiMapState = 1 THEN
		q_sState := 'RUN' ;
	ELSIF i_stInfoData.usiMapState = 2 THEN
		q_sState := 'STOP' ;
	ELSIF i_stInfoData.usiMapState = 3 THEN
		q_sState := 'SAFE' ;
	ELSE
		q_sState := 'Unknown' ;
END_IF

// THE 'safeOr' FB HAS NO DIAGNOSTIC BYTE TO DECODE!

END_FUNCTION_BLOCK

// POUs/ConnectionAndFb_Blocks/FBs/FB_InfoRS
(*=====================================================================
Beckhoff Automation LLC
Copyright 2015 All Rights Reserved
=======================================================================
Description: 
This Program has been supplied by Beckhoff Automation As-Is and is intended only as an example implementation. 
Functionality is not guaranteed. 
This Function Block reads status and error information known at time of creation of the TwinSAFE 'safeRs' 
function block.
---------------------------------------------------------------------------------------------------------------
History:
Date		Version			Author							Comment
---------------------------------------------------------------------------------------------------------------
07.08.15	0.10		Jason Erickson				Initial Library Creation.
07.20.15	0.11		Jason Ericskon				Added CoE Read for TwinSAFE Connection State.
08.28.15	0.20		Jason Erickson				Code optimization to eliminate timed data reads.
09.18.15	0.2.1		Jason Erickson				Added new error codes 0x6000 - 0x6002 and Connection Status
														to the AX5805.
*)
FUNCTION_BLOCK FB_InfoRS
VAR_INPUT
(* ***** Structure variables individually linked to the 'Function Block Info Data' of the EL69xx. ***** *)
	i_stInfoData: ST_SAFETY_FB ;
END_VAR
VAR_OUTPUT
// State of the TwinSAFE FB.
	q_sState: STRING ;
END_VAR

// Evaluate state of the TwinSAFE 'safeRs' FB.
IF i_stInfoData.usiMapState = 0 THEN
	q_sState := 'Undefined' ;
	ELSIF i_stInfoData.usiMapState = 2 THEN
		q_sState := 'STOP' ;
	ELSIF i_stInfoData.usiMapState = 3 THEN
		q_sState := 'SAFE' ;
	ELSIF i_stInfoData.usiMapState = 9 THEN
		q_sState := 'SET' ;
	ELSE
		q_sState := 'Unknown' ;
END_IF

// THE 'safeRs' FB HAS NO DIAGNOSTIC BYTE TO DECODE!

END_FUNCTION_BLOCK

// POUs/ConnectionAndFb_Blocks/FBs/FB_InfoSR
(*=====================================================================
Beckhoff Automation LLC
Copyright 2015 All Rights Reserved
=======================================================================
Description: 
This Program has been supplied by Beckhoff Automation As-Is and is intended only as an example implementation. 
Functionality is not guaranteed. 
This Function Block reads status and error information known at time of creation of the TwinSAFE 'safeSr' 
function block.
---------------------------------------------------------------------------------------------------------------
History:
Date		Version			Author							Comment
---------------------------------------------------------------------------------------------------------------
07.08.15	0.10		Jason Erickson				Initial Library Creation.
07.20.15	0.11		Jason Ericskon				Added CoE Read for TwinSAFE Connection State.
08.28.15	0.20		Jason Erickson				Code optimization to eliminate timed data reads.
09.18.15	0.2.1		Jason Erickson				Added new error codes 0x6000 - 0x6002 and Connection Status
														to the AX5805.
*)
FUNCTION_BLOCK FB_InfoSR
VAR_INPUT
(* ***** Structure variables individually linked to the 'Function Block Info Data' of the EL69xx. ***** *)
	i_stInfoData: ST_SAFETY_FB ;
END_VAR
VAR_OUTPUT
// State of the TwinSAFE FB.
	q_sState: STRING ;
END_VAR

// Evaluate state of the TwinSAFE 'safeSr' FB.
IF i_stInfoData.usiMapState = 0 THEN
	q_sState := 'Undefined' ;
	ELSIF i_stInfoData.usiMapState = 2 THEN
		q_sState := 'STOP' ;
	ELSIF i_stInfoData.usiMapState = 3 THEN
		q_sState := 'SAFE' ;
	ELSIF i_stInfoData.usiMapState = 9 THEN
		q_sState := 'SET' ;
	ELSE
		q_sState := 'Unknown' ;
END_IF

// THE 'safeSr' FB HAS NO DIAGNOSTIC BYTE TO DECODE!

END_FUNCTION_BLOCK

// POUs/ConnectionAndFb_Blocks/FBs/FB_InfoTOF
(*=====================================================================
Beckhoff Automation LLC
Copyright 2015 All Rights Reserved
=======================================================================
Description: 
This Program has been supplied by Beckhoff Automation As-Is and is intended only as an example implementation. 
Functionality is not guaranteed. 
This Function Block reads status and error information known at time of creation of the TwinSAFE 'safeTof' 
function block.
---------------------------------------------------------------------------------------------------------------
History:
Date		Version			Author							Comment
---------------------------------------------------------------------------------------------------------------
07.08.15	0.10		Jason Erickson				Initial Library Creation.
07.20.15	0.11		Jason Ericskon				Added CoE Read for TwinSAFE Connection State.
08.28.15	0.20		Jason Erickson				Code optimization to eliminate timed data reads.
09.18.15	0.2.1		Jason Erickson				Added new error codes 0x6000 - 0x6002 and Connection Status
														to the AX5805.
*)
FUNCTION_BLOCK FB_InfoTOF
VAR_INPUT
(* ***** Structure variables individually linked to the 'Function Block Info Data' of the EL69xx. ***** *)
	i_stInfoData: ST_SAFETY_FB ;
END_VAR
VAR_OUTPUT
// State of the TwinSAFE FB.
	q_sState: STRING ;
END_VAR

// Evaluate safeTof FB State
IF i_stInfoData.usiMapState = 0 THEN
	q_sState := 'Undefined' ;
	ELSIF i_stInfoData.usiMapState = 1 THEN
		q_sState := 'RUN' ;
	ELSIF i_stInfoData.usiMapState = 2 THEN
		q_sState := 'STOP' ;
	ELSIF i_stInfoData.usiMapState = 3 THEN
		q_sState := 'SAFE' ;
	ELSIF i_stInfoData.usiMapState = 8 THEN
		q_sState := 'DelayOut' ;
	ELSE
		q_sState := 'Unknown' ;
END_IF

// THE safeTof FB HAS NO DIAGNOSTIC BYTE TO DECODE!

END_FUNCTION_BLOCK

// POUs/ConnectionAndFb_Blocks/FBs/FB_InfoTON
(*=====================================================================
Beckhoff Automation LLC
Copyright 2015 All Rights Reserved
=======================================================================
Description: 
This Program has been supplied by Beckhoff Automation As-Is and is intended only as an example implementation. 
Functionality is not guaranteed. 
This Function Block reads status and error information known at time of creation of the TwinSAFE 'safeTon' 
function block.
---------------------------------------------------------------------------------------------------------------
History:
Date		Version			Author							Comment
---------------------------------------------------------------------------------------------------------------
07.08.15	0.10		Jason Erickson				Initial Library Creation.
07.20.15	0.11		Jason Ericskon				Added CoE Read for TwinSAFE Connection State.
08.28.15	0.20		Jason Erickson				Code optimization to eliminate timed data reads.
09.18.15	0.2.1		Jason Erickson				Added new error codes 0x6000 - 0x6002 and Connection Status
														to the AX5805.
*)
FUNCTION_BLOCK FB_InfoTON
VAR_INPUT
(* ***** Structure variables individually linked to the 'Function Block Info Data' of the EL69xx. ***** *)
	i_stInfoData: ST_SAFETY_FB ;
END_VAR
VAR_OUTPUT
// State of the TwinSAFE FB.
	q_sState: STRING ;
END_VAR

// Evaluate safeTon FB State
IF i_stInfoData.usiMapState = 0 THEN
	q_sState := 'Undefined' ;
	ELSIF i_stInfoData.usiMapState = 1 THEN
		q_sState := 'RUN' ;
	ELSIF i_stInfoData.usiMapState = 2 THEN
		q_sState := 'STOP' ;
	ELSIF i_stInfoData.usiMapState = 3 THEN
		q_sState := 'SAFE' ;
	ELSIF i_stInfoData.usiMapState = 9 THEN
		q_sState := 'DelayIn' ;
	ELSE
		q_sState := 'Unknown' ;
END_IF

// THE safeTon FB HAS NO DIAGNOSTIC BYTE TO DECODE!

END_FUNCTION_BLOCK

// POUs/ConnectionAndFb_Blocks/FBs/FB_InfoTwoHand
(*=====================================================================
Beckhoff Automation LLC
Copyright 2015 All Rights Reserved
=======================================================================
Description: 
This Program has been supplied by Beckhoff Automation As-Is and is intended only as an example implementation. 
Functionality is not guaranteed. 
This Function Block reads status and error information known at time of creation of the TwinSAFE 'safeTwohand' 
function block.
---------------------------------------------------------------------------------------------------------------
History:
Date		Version			Author							Comment
---------------------------------------------------------------------------------------------------------------
07.08.15	0.10		Jason Erickson				Initial Library Creation.
07.20.15	0.11		Jason Ericskon				Added CoE Read for TwinSAFE Connection State.
08.28.15	0.20		Jason Erickson				Code optimization to eliminate timed data reads.
09.18.15	0.2.1		Jason Erickson				Added new error codes 0x6000 - 0x6002 and Connection Status
														to the AX5805.
*)
FUNCTION_BLOCK FB_InfoTwoHand
VAR_INPUT
(* ***** Structure variables individually linked to the 'Function Block Info Data' of the EL69xx. ***** *)
	i_stInfoData: ST_SAFETY_FB ;
END_VAR
VAR_OUTPUT
// State of the TwinSAFE FB.
	q_sState: STRING ;
// Diagnostics of the TwinSAFE FB.
	q_sDiag: STRING ;
END_VAR

// Evaluate safeTwohand FB State.
IF i_stInfoData.usiMapState = 0 THEN
	q_sState := 'Undefined' ;
	ELSIF i_stInfoData.usiMapState = 1 THEN
		q_sState := 'RUN' ;
	ELSIF i_stInfoData.usiMapState = 2 THEN
		q_sState := 'STOP' ;
	ELSIF i_stInfoData.usiMapState = 3 THEN
		q_sState := 'SAFE' ;
	ELSIF i_stInfoData.usiMapState = 4 THEN
		q_sState := 'ERROR' ;
	ELSIF i_stInfoData.usiMapState = 5 THEN
		q_sState := 'RESET' ;
	ELSIF i_stInfoData.usiMapState = 6 THEN
		q_sState := 'START' ;
	ELSIF i_stInfoData.usiMapState = 11 THEN
		q_sState := '1BUTTON' ;
	ELSIF i_stInfoData.usiMapState = 12 THEN
		q_sState := '2BUTTON' ;
	ELSIF i_stInfoData.usiMapState = 13 THEN
		q_sState := 'RELEASE' ;
	ELSE
		q_sState := 'Unknown' ;
END_IF

// Evaluate safeTwohand FB Diagnostics
IF i_stInfoData.uiMapDiag = 0 THEN
	q_sDiag := 'No Error' ;
	ELSIF i_stInfoData.uiMapDiag = 1 THEN
		q_sDiag := 'Discrepancy Error Input Group 1' ;
	ELSIF i_stInfoData.uiMapDiag = 2 THEN
		q_sDiag := 'Discrepancy Error Input Group 2' ;
	ELSIF i_stInfoData.uiMapDiag = 4 THEN
		q_sDiag := 'Discrepancy Error Between Input Groups' ;
	ELSE
		q_sDiag := 'Unknown' ;
END_IF

END_FUNCTION_BLOCK

// POUs/ConnectionAndFb_Blocks/Project/FB_SafetyConnectionAX5805
(*=====================================================================
Beckhoff Automation LLC
Copyright 2015 All Rights Reserved
=======================================================================
Description: 
This Program has been supplied by Beckhoff Automation As-Is and is intended only as an example implementation. 
Functionality is not guaranteed. 
This Function Block reads status and error information known at time of creation of the TwinSAFE 'AX5805 TwinSAFE
Connection'.
---------------------------------------------------------------------------------------------------------------
History:
Date		Version			Author							Comment
---------------------------------------------------------------------------------------------------------------
07.08.15	0.10		Jason Erickson				Initial Library Creation.
07.20.15	0.11		Jason Ericskon				Added CoE Read for TwinSAFE Connection State.
08.28.15	0.20		Jason Erickson				Code optimization to eliminate timed data reads.
09.18.15	0.2.1		Jason Erickson				Added new error codes 0x6000 - 0x6002 and Connection Status
														to the AX5805.													
*)
FUNCTION_BLOCK FB_SafetyConnectionAX5805
VAR_INPUT
// Structure to bring status data into PLC.
	(* ***** Structure linked to the AX5805 'Connection Info Data' of the EL69xx. ***** *)
	i_stInfoData: ST_SAFETY_CONNECTION_AX5805;
END_VAR
VAR_OUTPUT
// State of the AX5805 TwinSAFE connection.
	q_sConnectionState: STRING;
	q_xModeErrorCh1: BOOL;
	q_sAX580xModeStateCh1: STRING;
	q_xModeErrorCh2: BOOL;
	q_sAX580xModeStateCh2: STRING;
// Connection Diagnostic of the AX5805.
	q_sDiag: STRING;
// Connection Input Status signals of the AX5805.
	q_bSafIn0: BYTE; // Input status of Channel 1 default motion functions and error.
	q_bSafIn1: BYTE; // Input status of Channel 1 USER CONFIGURED motion functions and error.
	q_bSafIn2: BYTE; // Input status of Channel 2 default motion functions and error.
	q_bSafIn3: BYTE; // Input status of Channel 2 USER CONFIGURED motion functions and error.
// Connection Output Status signals of the AX5805.
	q_bSafeOut0: BYTE; // Output status of Channel 1 default motion functions and error.
	q_bSafeOut1: BYTE; // Output status of Channel 1 USER CONFIGURED motion functions and error.
	q_bSafeOut2: BYTE; // Output status of Channel 2 default motion functions and error.
	q_bSafeOut3: BYTE; // Output status of Channel 2 USER CONFIGURED motion functions and error.
END_VAR

// Evaluate connection state of the TwinSAFE connection of the AX5805.

// Value 100 (0x64) 
	(* The Reset State: The reset state is used to re-initialize the Safety over 
		EtherCAT connection after the power-on or a Safety over EtherCAT communication error. *)
IF i_stInfoData.usiMapState = 100 THEN
	q_sConnectionState := 'Reset State' ;

// Value 101 (0x65) 
	(* The Session State: During the transition to or in the session state a session ID is transferred from
		the FSoE master to the SFoE slave, which in turn responds with its own session ID back to the FSoE master. *)
ELSIF i_stInfoData.usiMapState = 101 THEN
	q_sConnectionState := 'Session State' ;	

// Value 102 (0x66) 
	(* The Connection State: In the connection state a connection ID
		is transferred from the FSoE master to the FSoE slave. *)
ELSIF i_stInfoData.usiMapState = 102 THEN
	q_sConnectionState := 'Connection State' ;

// Value 103 (0x67) 
	(* The Parameter State: In the parameter state safe communication and device specific
		application parameters are transferred from the FSoE master to the FSoE slave. *)
ELSIF i_stInfoData.usiMapState = 103 THEN
	q_sConnectionState := 'Parameter State' ;

// Value 104 (0x68) 
	(* The Data Exchange State: In the data state FSoE cycles are transferred until
		either a communications error occurs or an FSoE node is stopped locally. *)
ELSIF i_stInfoData.usiMapState = 104 THEN
	q_sConnectionState := 'Data State' ;

// Value 105 (0x69) 
	(* The Shut Down State: In the shut down state the connection 
		was shutdown by one of the communication partners. *)
ELSIF i_stInfoData.usiMapState = 105 THEN
	q_sConnectionState := 'Shutdown State' ;

// Value is not between 100 and 105 so unknown state which is an error.
ELSE
	q_sConnectionState := 'Error' ;
END_IF

// Evaluate connection diagnostics of the TwinSAFE connection of the AX5805.

// Value		Description
// xxxx 0000	No Error
IF i_stInfoData.usiMapDiag = 0 THEN
	q_sDiag := 'No Error' ;

// Value		Description
// xxxx 0001	Invalid Command
ELSIF  i_stInfoData.usiMapDiag.0 = TRUE THEN
	q_sDiag := 'Invalid Command' ;

// Value		Description
// xxxx 0010	Unknown Command
ELSIF  i_stInfoData.usiMapDiag.1 = TRUE THEN
	q_sDiag := 'Unknown Command' ;

// Value		Description
// xxxx 0011	Invalid Connection ID
ELSIF  (i_stInfoData.usiMapDiag.0 AND i_stInfoData.usiMapDiag.1) = TRUE THEN
	q_sDiag := 'Invalid Connection-ID' ;

// Value		Description
// xxxx 0100	Invalid CRC	
ELSIF  i_stInfoData.usiMapDiag.2 = TRUE THEN
	q_sDiag := 'Invalid CRC' ;

// Value		Description
// xxxx 0101	Watchdog Time Elapsed
ELSIF  (i_stInfoData.usiMapDiag.0 AND i_stInfoData.usiMapDiag.2) = TRUE THEN
	q_sDiag := 'Watchdog Expired' ;
	
// Value		Description
// xxxx 0110	Invalid FSoE Address	
ELSIF  (i_stInfoData.usiMapDiag.1 AND i_stInfoData.usiMapDiag.2) = TRUE THEN
	q_sDiag := 'Invalid FSoE Address' ;

// Value		Description
// xxxx 0111	Invalid Data
ELSIF  (i_stInfoData.usiMapDiag.0 AND i_stInfoData.usiMapDiag.1 AND i_stInfoData.usiMapDiag.2) = TRUE THEN	
	q_sDiag := 'Invalid Data' ;
	
// Value		Description
// xxxx 1000	Invalid Communication Parameter Length
ELSIF  i_stInfoData.usiMapDiag.3 = TRUE THEN
	q_sDiag := 'Invalid Communication Parameter Length' ;

// Value		Description
// xxxx 1001	Invalid Communication Parameters
ELSIF  (i_stInfoData.usiMapDiag.0 AND i_stInfoData.usiMapDiag.3) = TRUE THEN
	q_sDiag := 'Invalid Commuication Parameters' ;

// Value		Description
// xxxx 1010	Invalid User Parameter Length
ELSIF  (i_stInfoData.usiMapDiag.1 AND i_stInfoData.usiMapDiag.3) = TRUE THEN
	q_sDiag := 'Invalid User Parameter Length' ;

// Value		Description
// xxxx 1011	Invalid User PArameters
ELSIF  (i_stInfoData.usiMapDiag.0 AND i_stInfoData.usiMapDiag.1 AND i_stInfoData.usiMapDiag.3) = TRUE THEN	
	q_sDiag := 'Invalid User Parameters' ;

// Value		Description
// xxxx 1100	FSoE Master Reset	
ELSIF  (i_stInfoData.usiMapDiag.2 AND i_stInfoData.usiMapDiag.3) = TRUE THEN
	q_sDiag := 'FSoE Master Reset' ;

// Value		Description
// 0001 xxxx	FSoE Slave Error Detected
ELSIF  i_stInfoData.usiMapDiag.4 = TRUE THEN
	q_sDiag := 'FSoE Slave Error Detected' ;

// Value		Description
// 0010 xxxx	FSoE Slave Reports Failsafe Value Active
ELSIF  i_stInfoData.usiMapDiag.5 = TRUE THEN
	q_sDiag := 'FSoE Slave Reports Failsafe Value Active' ;

// Value		Description
// 0100 xxxx	Connection is in Startup
ELSIF  i_stInfoData.usiMapDiag.6 = TRUE THEN
	q_sDiag := 'Connection Is In Startup' ;

// Value		Description
// 1000 xxxx	FSoE Master Reports Failsafe Value Active	
ELSIF  i_stInfoData.usiMapDiag.7 = TRUE THEN
	q_sDiag := 'FSoE Master Reports Failsafe Value Active' ;	

// Value		Description
//				Unknown Error
 				(* Something Not Specifically Annunciated Above.
 					possibly a combination OF errors are occuring. *)
ELSE	
	q_sDiag := 'Error' ;

END_IF

// Connection Info Data: Input Signals of the AX5805.
q_bSafIn0 := i_stInfoData.bInputSignals0 ; // Input status of Channel 1 default motion functions and error.
q_bSafIn1 := i_stInfoData.bInputSignals1 ; // Input status of Channel 1 USER CONFIGURED motion functions and error.
q_bSafIn2 := i_stInfoData.bInputSignals2 ; // Input status of Channel 2 default motion functions and error.
q_bSafIn3 := i_stInfoData.bInputSignals3 ; // Input status of Channel 2 USER CONFIGURED motion functions and error.
// Connection Info Data: Output Signals of the AX5805.
q_bSafeOut0 := i_stInfoData.bOutputSignals0 ; // Output status of Channel 1 default motion functions and error.
q_bSafeOut1 := i_stInfoData.bOutputSignals1 ; // Output status of Channel 1 USER CONFIGURED motion functions and error.
q_bSafeOut2 := i_stInfoData.bOutputSignals2 ; // Output status of Channel 2 default motion functions and error.
q_bSafeOut3 := i_stInfoData.bOutputSignals3 ; // Output status of Channel 2 USER CONFIGURED motion functions and error.

// Bit 7 is the AX5805 Connection Error Status channel 1.
IF i_stInfoData.bInputSignals0.7 THEN
	q_xModeErrorCh1 := TRUE;
ELSIF NOT i_stInfoData.bInputSignals0.7 THEN
	q_xModeErrorCh1 := FALSE;
END_IF

// Bit 0-6 is the Activation Status of the AX5805 motion functions channel 1.
IF i_stInfoData.bInputSignals0.0 THEN
	q_sAX580xModeStateCh1 := 'STO is set Ch1.';
ELSIF i_stInfoData.bInputSignals0.1 THEN
	q_sAX580xModeStateCh1 := 'SS1 is set Ch1.';
ELSIF i_stInfoData.bInputSignals0.2 THEN
	q_sAX580xModeStateCh1 := 'SS2 is set Ch1.';
ELSIF i_stInfoData.bInputSignals0.3 THEN
	q_sAX580xModeStateCh1 := 'SOS is set Ch1.';
ELSIF i_stInfoData.bInputSignals0.4 THEN
	q_sAX580xModeStateCh1 := 'SSR is set Ch1.';
ELSIF i_stInfoData.bInputSignals0.5 THEN
	q_sAX580xModeStateCh1 := 'SDIp is set Ch1.';
ELSIF i_stInfoData.bInputSignals0.6 THEN
	q_sAX580xModeStateCh1 := 'SDIn is set Ch1.';
ELSE
	q_sAX580xModeStateCh1 := 'RUN.';
END_IF

// Bit 7 is the AX5805 Connection Error Status channel 2.
IF i_stInfoData.bInputSignals2.7 THEN
	q_xModeErrorCh2 := TRUE;
ELSIF NOT i_stInfoData.bInputSignals2.7 THEN
	q_xModeErrorCh2 := FALSE;
END_IF

// Bit 0-6 is the Activation Status of the AX5805 motion functions channel 2.
IF i_stInfoData.bInputSignals2.0 THEN
	q_sAX580xModeStateCh2 := 'STO is set Ch2.';
ELSIF i_stInfoData.bInputSignals2.1 THEN
	q_sAX580xModeStateCh2 := 'SS1 is set Ch2.';
ELSIF i_stInfoData.bInputSignals2.2 THEN
	q_sAX580xModeStateCh2 := 'SS2 is set Ch2.';
ELSIF i_stInfoData.bInputSignals2.3 THEN
	q_sAX580xModeStateCh2 := 'SOS is set Ch2.';
ELSIF i_stInfoData.bInputSignals2.4 THEN
	q_sAX580xModeStateCh2 := 'SSR is set Ch2.';
ELSIF i_stInfoData.bInputSignals2.5 THEN
	q_sAX580xModeStateCh2 := 'SDIp is set Ch2.';
ELSIF i_stInfoData.bInputSignals2.6 THEN
	q_sAX580xModeStateCh2 := 'SDIn is set Ch2.';
ELSE
	q_sAX580xModeStateCh2 := 'RUN.';
END_IF

END_FUNCTION_BLOCK

// POUs/ConnectionAndFb_Blocks/Project/FB_SafetyConnectionEK1914
(*=====================================================================
Beckhoff Automation LLC
Copyright 2015 All Rights Reserved
=======================================================================
Description: 
This Program has been supplied by Beckhoff Automation As-Is and is intended only as an example implementation. 
Functionality is not guaranteed. 
This Function Block reads status and error information known at time of creation of the TwinSAFE 'EK1914 TwinSAFE
Connection'.
---------------------------------------------------------------------------------------------------------------
History:
Date		Version			Author							Comment
---------------------------------------------------------------------------------------------------------------
07.08.15	0.10		Jason Erickson				Initial Library Creation.
07.20.15	0.11		Jason Ericskon				Added CoE Read for TwinSAFE Connection State.
08.28.15	0.20		Jason Erickson				Code optimization to eliminate timed data reads.
09.18.15	0.2.1		Jason Erickson				Added new error codes 0x6000 - 0x6002 and Connection Status
														to the AX5805.													
*)
FUNCTION_BLOCK FB_SafetyConnectionEK1914
VAR_INPUT
// Structure to bring status data into PLC.
	(* ***** Structure linked to the EK1914 'Connection Info Data' of the EL69xx. ***** *)
	i_stInfoData: ST_SAFETY_CONNECTION_EK1914;
END_VAR
VAR_OUTPUT
// State of the EK1914 TwinSAFE connection.
	q_sState: STRING;
// Connection Diagnostic of the EK1914.
	q_sDiag: STRING;
// Input Signals of the EK1914.
	q_xSafIn1: BOOL;
	q_xSafIn2: BOOL;
	q_xSafeOut1: BOOL;
	q_xSafeOut2: BOOL;
END_VAR

// Evaluate connection state of the TwinSAFE connection of the EK1914.

// Value 100 (0x64) 
	(* The Reset State: The reset state is used to re-initialize the Safety over 
		EtherCAT connection after the power-on or a Safety over EtherCAT communication error. *)
IF i_stInfoData.usiMapState = 100 THEN
	q_sState := 'Reset State' ;

// Value 101 (0x65) 
	(* The Session State: During the transition to or in the session state a session ID is transferred from
		the FSoE master to the SFoE slave, which in turn responds with its own session ID back to the FSoE master. *)
ELSIF i_stInfoData.usiMapState = 101 THEN
	q_sState := 'Session State' ;	

// Value 102 (0x66) 
	(* The Connection State: In the connection state a connection ID
		is transferred from the FSoE master to the FSoE slave. *)
ELSIF i_stInfoData.usiMapState = 102 THEN
	q_sState := 'Connection State' ;

// Value 103 (0x67) 
	(* The Parameter State: In the parameter state safe communication and device specific
		application parameters are transferred from the FSoE master to the FSoE slave. *)
ELSIF i_stInfoData.usiMapState = 103 THEN
	q_sState := 'Parameter State' ;

// Value 104 (0x68) 
	(* The Data Exchange State: In the data state FSoE cycles are transferred until
		either a communications error occurs or an FSoE node is stopped locally. *)
ELSIF i_stInfoData.usiMapState = 104 THEN
	q_sState := 'Data State' ;

// Value 105 (0x69) 
	(* The Shut Down State: In the shut down state the connection 
		was shutdown by one of the communication partners. *)
ELSIF i_stInfoData.usiMapState = 105 THEN
	q_sState := 'Shutdown State' ;

// Value is not between 100 and 105 so unknown state which is an error.
ELSE
	q_sState := 'Error' ;
END_IF

// Evaluate connection diagnostics of the TwinSAFE connection of the EK1914.

// Value		Description
// xxxx 0000	No Error
IF i_stInfoData.usiMapDiag = 0 THEN
	q_sDiag := 'No Error' ;

// Value		Description
// xxxx 0001	Invalid Command
ELSIF  i_stInfoData.usiMapDiag.0 = TRUE THEN
	q_sDiag := 'Invalid Command' ;

// Value		Description
// xxxx 0010	Unknown Command
ELSIF  i_stInfoData.usiMapDiag.1 = TRUE THEN
	q_sDiag := 'Unknown Command' ;

// Value		Description
// xxxx 0011	Invalid Connection ID
ELSIF  (i_stInfoData.usiMapDiag.0 AND i_stInfoData.usiMapDiag.1) = TRUE THEN
	q_sDiag := 'Invalid Connection-ID' ;

// Value		Description
// xxxx 0100	Invalid CRC	
ELSIF  i_stInfoData.usiMapDiag.2 = TRUE THEN
	q_sDiag := 'Invalid CRC' ;

// Value		Description
// xxxx 0101	Watchdog Time Elapsed
ELSIF  (i_stInfoData.usiMapDiag.0 AND i_stInfoData.usiMapDiag.2) = TRUE THEN
	q_sDiag := 'Watchdog Expired' ;
	
// Value		Description
// xxxx 0110	Invalid FSoE Address	
ELSIF  (i_stInfoData.usiMapDiag.1 AND i_stInfoData.usiMapDiag.2) = TRUE THEN
	q_sDiag := 'Invalid FSoE Address' ;

// Value		Description
// xxxx 0111	Invalid Data
ELSIF  (i_stInfoData.usiMapDiag.0 AND i_stInfoData.usiMapDiag.1 AND i_stInfoData.usiMapDiag.2) = TRUE THEN	
	q_sDiag := 'Invalid Data' ;
	
// Value		Description
// xxxx 1000	Invalid Communication Parameter Length
ELSIF  i_stInfoData.usiMapDiag.3 = TRUE THEN
	q_sDiag := 'Invalid Communication Parameter Length' ;

// Value		Description
// xxxx 1001	Invalid Communication Parameters
ELSIF  (i_stInfoData.usiMapDiag.0 AND i_stInfoData.usiMapDiag.3) = TRUE THEN
	q_sDiag := 'Invalid Commuication Parameters' ;

// Value		Description
// xxxx 1010	Invalid User Parameter Length
ELSIF  (i_stInfoData.usiMapDiag.1 AND i_stInfoData.usiMapDiag.3) = TRUE THEN
	q_sDiag := 'Invalid User Parameter Length' ;

// Value		Description
// xxxx 1011	Invalid User PArameters
ELSIF  (i_stInfoData.usiMapDiag.0 AND i_stInfoData.usiMapDiag.1 AND i_stInfoData.usiMapDiag.3) = TRUE THEN	
	q_sDiag := 'Invalid User Parameters' ;

// Value		Description
// xxxx 1100	FSoE Master Reset	
ELSIF  (i_stInfoData.usiMapDiag.2 AND i_stInfoData.usiMapDiag.3) = TRUE THEN
	q_sDiag := 'FSoE Master Reset' ;

// Value		Description
// 0001 xxxx	FSoE Slave Error Detected
ELSIF  i_stInfoData.usiMapDiag.4 = TRUE THEN
	q_sDiag := 'FSoE Slave Error Detected' ;

// Value		Description
// 0010 xxxx	FSoE Slave Reports Failsafe Value Active
ELSIF  i_stInfoData.usiMapDiag.5 = TRUE THEN
	q_sDiag := 'FSoE Slave Reports Failsafe Value Active' ;

// Value		Description
// 0100 xxxx	Connection is in Startup
ELSIF  i_stInfoData.usiMapDiag.6 = TRUE THEN
	q_sDiag := 'Connection Is In Startup' ;

// Value		Description
// 1000 xxxx	FSoE Master Reports Failsafe Value Active	
ELSIF  i_stInfoData.usiMapDiag.7 = TRUE THEN
	q_sDiag := 'FSoE Master Reports Failsafe Value Active' ;	

// Value		Description
//				Unknown Error
 				(* Something Not Specifically Annunciated Above.
 					possibly a combination OF errors are occuring. *)
ELSE	
	q_sDiag := 'Error' ;

END_IF

// Input Signals of the EK1914.
q_xSafIn1 := i_stInfoData.bInputSignals.0 ;
q_xSafIn2 := i_stInfoData.bInputSignals.1 ;
// Output Signals of the EK1914.
q_xSafeOut1 := i_stInfoData.bOutputSignals.0 ;
q_xSafeOut2 := i_stInfoData.bOutputSignals.1 ;

END_FUNCTION_BLOCK

// POUs/ConnectionAndFb_Blocks/Project/FB_SafetyConnectionEL1904
(*=====================================================================
Beckhoff Automation LLC
Copyright 2015 All Rights Reserved
=======================================================================
Description: 
This Program has been supplied by Beckhoff Automation As-Is and is intended only as an example implementation. 
Functionality is not guaranteed. 
This Function Block reads status and error information known at time of creation of the TwinSAFE 'EL1904 TwinSAFE
Connection'.
---------------------------------------------------------------------------------------------------------------
History:
Date		Version			Author							Comment
---------------------------------------------------------------------------------------------------------------
07.08.15	0.10		Jason Erickson				Initial Library Creation.
07.20.15	0.11		Jason Ericskon				Added CoE Read for TwinSAFE Connection State.
08.28.15	0.20		Jason Erickson				Code optimization to eliminate timed data reads.
09.18.15	0.2.1		Jason Erickson				Added new error codes 0x6000 - 0x6002 and Connection Status
														to the AX5805.
*)
FUNCTION_BLOCK FB_SafetyConnectionEL1904
VAR_INPUT
// Structure to bring status data into PLC.
	(* ***** Structure linked to the EL1904 'Connection Info Data' of the EL69xx. ***** *)
	i_stInfoData: ST_SAFETY_CONNECTION_EL1904;
END_VAR
VAR_OUTPUT
// State of the EL1904 TwinSAFE connection.
	q_sState: STRING;
// Connection Diagnostic of the EL1904.
	q_sDiag: STRING;
// Input Signals of the EL1904.
	q_xChannel1: BOOL;
	q_xChannel2: BOOL;
	q_xChannel3: BOOL;
	q_xChannel4: BOOL;
END_VAR

// Evaluate connection state of the TwinSAFE connection of the EL1904.

// Value 100 (0x64) 
	(* The Reset State: The reset state is used to re-initialize the Safety over 
		EtherCAT connection after the power-on or a Safety over EtherCAT communication error. *)
IF i_stInfoData.usiMapState = 100 THEN
	q_sState := 'Reset State' ;

// Value 101 (0x65) 
	(* The Session State: During the transition to or in the session state a session ID is transferred from
		the FSoE master to the SFoE slave, which in turn responds with its own session ID back to the FSoE master. *)
ELSIF i_stInfoData.usiMapState = 101 THEN
	q_sState := 'Session State' ;	

// Value 102 (0x66) 
	(* The Connection State: In the connection state a connection ID
		is transferred from the FSoE master to the FSoE slave. *)
ELSIF i_stInfoData.usiMapState = 102 THEN
	q_sState := 'Connection State' ;

// Value 103 (0x67) 
	(* The Parameter State: In the parameter state safe communication and device specific
		application parameters are transferred from the FSoE master to the FSoE slave. *)
ELSIF i_stInfoData.usiMapState = 103 THEN
	q_sState := 'Parameter State' ;

// Value 104 (0x68) 
	(* The Data Exchange State: In the data state FSoE cycles are transferred until
		either a communications error occurs or an FSoE node is stopped locally. *)
ELSIF i_stInfoData.usiMapState = 104 THEN
	q_sState := 'Data State' ;

// Value 105 (0x69) 
	(* The Shut Down State: In the shut down state the connection 
		was shutdown by one of the communication partners. *)
ELSIF i_stInfoData.usiMapState = 105 THEN
	q_sState := 'Shutdown State' ;

// Value is not between 100 and 105 so unknown state which is an error.
ELSE
	q_sState := 'Error' ;
END_IF

// Evaluate connection diagnostics of the TwinSAFE connection of the EL1904.

// Value		Description
// xxxx 0000	No Error
IF i_stInfoData.usiMapDiag = 0 THEN
	q_sDiag := 'No Error' ;

// Value		Description
// xxxx 0001	Invalid Command
ELSIF  i_stInfoData.usiMapDiag.0 = TRUE THEN
	q_sDiag := 'Invalid Command' ;

// Value		Description
// xxxx 0010	Unknown Command
ELSIF  i_stInfoData.usiMapDiag.1 = TRUE THEN
	q_sDiag := 'Unknown Command' ;

// Value		Description
// xxxx 0011	Invalid Connection ID
ELSIF  (i_stInfoData.usiMapDiag.0 AND i_stInfoData.usiMapDiag.1) = TRUE THEN
	q_sDiag := 'Invalid Connection-ID' ;

// Value		Description
// xxxx 0100	Invalid CRC	
ELSIF  i_stInfoData.usiMapDiag.2 = TRUE THEN
	q_sDiag := 'Invalid CRC' ;

// Value		Description
// xxxx 0101	Watchdog Time Elapsed
ELSIF  (i_stInfoData.usiMapDiag.0 AND i_stInfoData.usiMapDiag.2) = TRUE THEN
	q_sDiag := 'Watchdog Expired' ;
	
// Value		Description
// xxxx 0110	Invalid FSoE Address	
ELSIF  (i_stInfoData.usiMapDiag.1 AND i_stInfoData.usiMapDiag.2) = TRUE THEN
	q_sDiag := 'Invalid FSoE Address' ;

// Value		Description
// xxxx 0111	Invalid Data
ELSIF  (i_stInfoData.usiMapDiag.0 AND i_stInfoData.usiMapDiag.1 AND i_stInfoData.usiMapDiag.2) = TRUE THEN	
	q_sDiag := 'Invalid Data' ;
	
// Value		Description
// xxxx 1000	Invalid Communication Parameter Length
ELSIF  i_stInfoData.usiMapDiag.3 = TRUE THEN
	q_sDiag := 'Invalid Communication Parameter Length' ;

// Value		Description
// xxxx 1001	Invalid Communication Parameters
ELSIF  (i_stInfoData.usiMapDiag.0 AND i_stInfoData.usiMapDiag.3) = TRUE THEN
	q_sDiag := 'Invalid Commuication Parameters' ;

// Value		Description
// xxxx 1010	Invalid User Parameter Length
ELSIF  (i_stInfoData.usiMapDiag.1 AND i_stInfoData.usiMapDiag.3) = TRUE THEN
	q_sDiag := 'Invalid User Parameter Length' ;

// Value		Description
// xxxx 1011	Invalid User PArameters
ELSIF  (i_stInfoData.usiMapDiag.0 AND i_stInfoData.usiMapDiag.1 AND i_stInfoData.usiMapDiag.3) = TRUE THEN	
	q_sDiag := 'Invalid User Parameters' ;

// Value		Description
// xxxx 1100	FSoE Master Reset	
ELSIF  (i_stInfoData.usiMapDiag.2 AND i_stInfoData.usiMapDiag.3) = TRUE THEN
	q_sDiag := 'FSoE Master Reset' ;

// Value		Description
// 0001 xxxx	FSoE Slave Error Detected
ELSIF  i_stInfoData.usiMapDiag.4 = TRUE THEN
	q_sDiag := 'FSoE Slave Error Detected' ;

// Value		Description
// 0010 xxxx	FSoE Slave Reports Failsafe Value Active
ELSIF  i_stInfoData.usiMapDiag.5 = TRUE THEN
	q_sDiag := 'FSoE Slave Reports Failsafe Value Active' ;

// Value		Description
// 0100 xxxx	Connection is in Startup
ELSIF  i_stInfoData.usiMapDiag.6 = TRUE THEN
	q_sDiag := 'Connection Is In Startup' ;

// Value		Description
// 1000 xxxx	FSoE Master Reports Failsafe Value Active	
ELSIF  i_stInfoData.usiMapDiag.7 = TRUE THEN
	q_sDiag := 'FSoE Master Reports Failsafe Value Active' ;	

// Value		Description
//				Unknown Error
 				(* Something Not Specifically Annunciated Above.
 					possibly a combination OF errors are occuring. *)
ELSE	
	q_sDiag := 'Error' ;

END_IF


// Input Signals of the EL1904.
q_xChannel1 := i_stInfoData.bInputSignals.0 ;
q_xChannel2 := i_stInfoData.bInputSignals.1 ;
q_xChannel3 := i_stInfoData.bInputSignals.2 ;
q_xChannel4 := i_stInfoData.bInputSignals.3 ;

END_FUNCTION_BLOCK

// POUs/ConnectionAndFb_Blocks/Project/FB_SafetyConnectionEL2904
(*=====================================================================
Beckhoff Automation LLC
Copyright 2015 All Rights Reserved
=======================================================================
Description: 
This Program has been supplied by Beckhoff Automation As-Is and is intended only as an example implementation. 
Functionality is not guaranteed. 
This Function Block reads status and error information known at time of creation of the TwinSAFE 'EL2904 TwinSAFE
Connection'.
---------------------------------------------------------------------------------------------------------------
History:
Date		Version			Author							Comment
---------------------------------------------------------------------------------------------------------------
07.08.15	0.10		Jason Erickson				Initial Library Creation.
07.20.15	0.11		Jason Ericskon				Added CoE Read for TwinSAFE Connection State.
08.28.15	0.20		Jason Erickson				Code optimization to eliminate timed data reads.
09.18.15	0.2.1		Jason Erickson				Added new error codes 0x6000 - 0x6002 and Connection Status
														to the AX5805.
*)
FUNCTION_BLOCK FB_SafetyConnectionEL2904
VAR_INPUT
// Structure to bring status data into PLC.
	(* ***** Structure linked to the EL2904 'Connection Info Data' of the EL69xx. ***** *)
	i_stInfoData: ST_SAFETY_CONNECTION_EL2904;
END_VAR
VAR_OUTPUT
// State of the EL2904 TwinSAFE connection.
	q_sState: STRING;
// Connection Diagnostic of the EL2904.
	q_sDiag: STRING;
// Output Signals of the EL2904.
	q_xChannel1: BOOL;
	q_xChannel2: BOOL;
	q_xChannel3: BOOL;
	q_xChannel4: BOOL;
END_VAR

// Evaluate connection state of the TwinSAFE connection of the EL2904.

// Value 100 (0x64) 
	(* The Reset State: The reset state is used to re-initialize the Safety over EtherCAT 
		connection after the power-on or a Safety over EtherCAT communication error. *)
IF i_stInfoData.usiMapState = 100 THEN
	q_sState := 'Reset State' ;

// Value 101 (0x65) 
	(* The Session State: During the transition to or in the session state a session ID is transferred from the  
		FSoE master to the SFoE slave, which in turn responds with its own session ID back to the FSoE master. *)
ELSIF i_stInfoData.usiMapState = 101 THEN
	q_sState := 'Session State' ;	

// Value 102 (0x66) 
	(* The Connection State: In the connection state a connection ID 
		 is transferred from the FSoE master to the FSoE slave. *)
ELSIF i_stInfoData.usiMapState = 102 THEN
	q_sState := 'Connection State' ;

// Value 103 (0x67) 
	(* The Parameter State: In the parameter state safe communication and device specific 
		application parameters are transferred from the FSoE master to the FSoE slave.*)
ELSIF i_stInfoData.usiMapState = 103 THEN
	q_sState := 'Parameter State' ;

// Value 104 (0x68) 
	(* The Data Exchange State: In the data state FSoE cycles are transferred until  
		either a communications error occurs or an FSoE node is stopped locally. *)
ELSIF i_stInfoData.usiMapState = 104 THEN
	q_sState := 'Data State' ;

// Value 105 (0x69) 
	(* The Shut Down State: In the shut down state the connection 
		was shutdown by one of the communication partners. *)
ELSIF i_stInfoData.usiMapState = 105 THEN
	q_sState := 'Shutdown State' ;

// Value is not between 100 and 105 so unknown state which is an error
ELSE
	q_sState := 'Error' ;
END_IF

// Evaluate connection diagnostics of the TwinSAFE connection of the EL2904.

// Value		Description
// xxxx 0000	No Error
IF i_stInfoData.usiMapDiag = 0 THEN
	q_sDiag := 'No Error' ;

// Value		Description
// xxxx 0001	Invalid Command
ELSIF  i_stInfoData.usiMapDiag.0 = TRUE THEN
	q_sDiag := 'Invalid Command' ;

// Value		Description
// xxxx 0010	Unknown Command
ELSIF  i_stInfoData.usiMapDiag.1 = TRUE THEN
	q_sDiag := 'Unknown Command' ;

// Value		Description
// xxxx 0011	Invalid Connection ID
ELSIF  (i_stInfoData.usiMapDiag.0 AND i_stInfoData.usiMapDiag.1) = TRUE THEN
	q_sDiag := 'Invalid Connection-ID' ;

// Value		Description
// xxxx 0100	Invalid CRC
ELSIF  i_stInfoData.usiMapDiag.2 = TRUE THEN
	q_sDiag := 'Invalid CRC' ;

// Value		Description
// xxxx 0101	Watchdog Time Elapsed
ELSIF  (i_stInfoData.usiMapDiag.0 AND i_stInfoData.usiMapDiag.2) = TRUE THEN
	q_sDiag := 'Watchdog Expired' ;
	
// Value		Description
// xxxx 0110	Invalid FSoE Address	
ELSIF  (i_stInfoData.usiMapDiag.1 AND i_stInfoData.usiMapDiag.2) = TRUE THEN
	q_sDiag := 'Invalid FSoE Address' ;

// Value		Description
// xxxx 0111	Invalid Data
ELSIF  (i_stInfoData.usiMapDiag.0 AND i_stInfoData.usiMapDiag.1 AND i_stInfoData.usiMapDiag.2) = TRUE THEN	
	q_sDiag := 'Invalid Data' ;
	
// Value		Description
// xxxx 1000	Invalid Communication Parameter Length
ELSIF  i_stInfoData.usiMapDiag.3 = TRUE THEN
	q_sDiag := 'Invalid Communication Parameter Length' ;

// Value		Description
// xxxx 1001	Invalid Communication Parameters
ELSIF  (i_stInfoData.usiMapDiag.0 AND i_stInfoData.usiMapDiag.3) = TRUE THEN
	q_sDiag := 'Invalid Commuication Parameters' ;

// Value		Description
// xxxx 1010	Invalid User Parameter Length
ELSIF  (i_stInfoData.usiMapDiag.1 AND i_stInfoData.usiMapDiag.3) = TRUE THEN
	q_sDiag := 'Invalid User Parameter Length' ;

// Value		Description
// xxxx 1011	Invalid User PArameters
ELSIF  (i_stInfoData.usiMapDiag.0 AND i_stInfoData.usiMapDiag.1 AND i_stInfoData.usiMapDiag.3) = TRUE THEN	
	q_sDiag := 'Invalid User Parameters' ;

// Value		Description
// xxxx 1100	FSoE Master Reset	
ELSIF  (i_stInfoData.usiMapDiag.2 AND i_stInfoData.usiMapDiag.3) = TRUE THEN
	q_sDiag := 'FSoE Master Reset' ;

// Value		Description
// 0001 xxxx	FSoE Slave Error Detected
ELSIF  i_stInfoData.usiMapDiag.4 = TRUE THEN
	q_sDiag := 'FSoE Slave Error Detected' ;

// Value		Description
// 0010 xxxx	FSoE Slave Reports Failsafe Value Active
ELSIF  i_stInfoData.usiMapDiag.5 = TRUE THEN
	q_sDiag := 'FSoE Slave Reports Failsafe Value Active' ;

// Value		Description
// 0100 xxxx	Connection is in Startup
ELSIF  i_stInfoData.usiMapDiag.6 = TRUE THEN
	q_sDiag := 'Connection Is In Startup' ;

// Value		Description
// 1000 xxxx	FSoE Master Reports Failsafe Value Active	
ELSIF  i_stInfoData.usiMapDiag.7 = TRUE THEN
	q_sDiag := 'FSoE Master Reports Failsafe Value Active' ;	

// Value		Description
//				Unknown Error
 				(* Something Not Specifically Annunciated Above.
 					possibly a combination OF errors are occuring. *)
ELSE	
	q_sDiag := 'Error' ;

END_IF

// Output Signals of the EL2904.
q_xChannel1 := i_stInfoData.bOutputSignals.0 ;
q_xChannel2 := i_stInfoData.bOutputSignals.1 ;
q_xChannel3 := i_stInfoData.bOutputSignals.2 ;
q_xChannel4 := i_stInfoData.bOutputSignals.3 ;

END_FUNCTION_BLOCK

// POUs/ConnectionAndFb_Blocks/Project/FB_SafetyConnectionEP1908
(*=====================================================================
Beckhoff Automation LLC
Copyright 2015 All Rights Reserved
=======================================================================
Description: 
This Program has been supplied by Beckhoff Automation As-Is and is intended only as an example implementation. 
Functionality is not guaranteed. 
This Function Block reads status and error information known at time of creation of the TwinSAFE 'EP1908 TwinSAFE
Connection'.
---------------------------------------------------------------------------------------------------------------
History:
Date		Version			Author							Comment
---------------------------------------------------------------------------------------------------------------
07.08.15	0.10		Jason Erickson				Initial Library Creation.
07.20.15	0.11		Jason Ericskon				Added CoE Read for TwinSAFE Connection State.
08.28.15	0.20		Jason Erickson				Code optimization to eliminate timed data reads.
09.18.15	0.2.1		Jason Erickson				Added new error codes 0x6000 - 0x6002 and Connection Status
														to the AX5805.
*)
FUNCTION_BLOCK FB_SafetyConnectionEP1908
VAR_INPUT
// Structure to bring status data into PLC.
	(* ***** Structure linked to the EP1908 'Connection Info Data' of the EL69xx. ***** *)
	i_stInfoData: ST_SAFETY_CONNECTION_EP1908;
END_VAR
VAR_OUTPUT
// State of the EP1908 TwinSAFE connection.
	q_sState: STRING;
// Connection Diagnostic of the EP1908.
	q_sDiag: STRING;
// Input Signals of the EP1908.
	q_xSafIn1: BOOL;
	q_xSafIn2: BOOL;
	q_xSafIn3: BOOL;
	q_xSafIn4: BOOL;
	q_xSafIn5: BOOL;
	q_xSafIn6: BOOL;
	q_xSafIn7: BOOL;
	q_xSafIn8: BOOL;
END_VAR

// Evaluate connection state of the TwinSAFE connection of the EP1908.

// Value 100 (0x64) 
	(* The Reset State: The reset state is used to re-initialize the Safety over 
		EtherCAT connection after the power-on or a Safety over EtherCAT communication error. *)
IF i_stInfoData.usiMapState = 100 THEN
	q_sState := 'Reset State' ;

// Value 101 (0x65) 
	(* The Session State: During the transition to or in the session state a session ID is transferred from
		the FSoE master to the SFoE slave, which in turn responds with its own session ID back to the FSoE master. *)
ELSIF i_stInfoData.usiMapState = 101 THEN
	q_sState := 'Session State' ;	

// Value 102 (0x66) 
	(* The Connection State: In the connection state a connection ID
		is transferred from the FSoE master to the FSoE slave. *)
ELSIF i_stInfoData.usiMapState = 102 THEN
	q_sState := 'Connection State' ;

// Value 103 (0x67) 
	(* The Parameter State: In the parameter state safe communication and device specific
		application parameters are transferred from the FSoE master to the FSoE slave. *)
ELSIF i_stInfoData.usiMapState = 103 THEN
	q_sState := 'Parameter State' ;

// Value 104 (0x68) 
	(* The Data Exchange State: In the data state FSoE cycles are transferred until
		either a communications error occurs or an FSoE node is stopped locally. *)
ELSIF i_stInfoData.usiMapState = 104 THEN
	q_sState := 'Data State' ;

// Value 105 (0x69) 
	(* The Shut Down State: In the shut down state the connection 
		was shutdown by one of the communication partners. *)
ELSIF i_stInfoData.usiMapState = 105 THEN
	q_sState := 'Shutdown State' ;

// Value is not between 100 and 105 so unknown state which is an error.
ELSE
	q_sState := 'Error' ;
END_IF

// Evaluate connection diagnostics of the TwinSAFE connection of the EP1908.

// Value		Description
// xxxx 0000	No Error
IF i_stInfoData.usiMapDiag = 0 THEN
	q_sDiag := 'No Error' ;

// Value		Description
// xxxx 0001	Invalid Command
ELSIF  i_stInfoData.usiMapDiag.0 = TRUE THEN
	q_sDiag := 'Invalid Command' ;

// Value		Description
// xxxx 0010	Unknown Command
ELSIF  i_stInfoData.usiMapDiag.1 = TRUE THEN
	q_sDiag := 'Unknown Command' ;

// Value		Description
// xxxx 0011	Invalid Connection ID
ELSIF  (i_stInfoData.usiMapDiag.0 AND i_stInfoData.usiMapDiag.1) = TRUE THEN
	q_sDiag := 'Invalid Connection-ID' ;

// Value		Description
// xxxx 0100	Invalid CRC	
ELSIF  i_stInfoData.usiMapDiag.2 = TRUE THEN
	q_sDiag := 'Invalid CRC' ;

// Value		Description
// xxxx 0101	Watchdog Time Elapsed
ELSIF  (i_stInfoData.usiMapDiag.0 AND i_stInfoData.usiMapDiag.2) = TRUE THEN
	q_sDiag := 'Watchdog Expired' ;
	
// Value		Description
// xxxx 0110	Invalid FSoE Address	
ELSIF  (i_stInfoData.usiMapDiag.1 AND i_stInfoData.usiMapDiag.2) = TRUE THEN
	q_sDiag := 'Invalid FSoE Address' ;

// Value		Description
// xxxx 0111	Invalid Data
ELSIF  (i_stInfoData.usiMapDiag.0 AND i_stInfoData.usiMapDiag.1 AND i_stInfoData.usiMapDiag.2) = TRUE THEN	
	q_sDiag := 'Invalid Data' ;
	
// Value		Description
// xxxx 1000	Invalid Communication Parameter Length
ELSIF  i_stInfoData.usiMapDiag.3 = TRUE THEN
	q_sDiag := 'Invalid Communication Parameter Length' ;

// Value		Description
// xxxx 1001	Invalid Communication Parameters
ELSIF  (i_stInfoData.usiMapDiag.0 AND i_stInfoData.usiMapDiag.3) = TRUE THEN
	q_sDiag := 'Invalid Commuication Parameters' ;

// Value		Description
// xxxx 1010	Invalid User Parameter Length
ELSIF  (i_stInfoData.usiMapDiag.1 AND i_stInfoData.usiMapDiag.3) = TRUE THEN
	q_sDiag := 'Invalid User Parameter Length' ;

// Value		Description
// xxxx 1011	Invalid User PArameters
ELSIF  (i_stInfoData.usiMapDiag.0 AND i_stInfoData.usiMapDiag.1 AND i_stInfoData.usiMapDiag.3) = TRUE THEN	
	q_sDiag := 'Invalid User Parameters' ;

// Value		Description
// xxxx 1100	FSoE Master Reset	
ELSIF  (i_stInfoData.usiMapDiag.2 AND i_stInfoData.usiMapDiag.3) = TRUE THEN
	q_sDiag := 'FSoE Master Reset' ;

// Value		Description
// 0001 xxxx	FSoE Slave Error Detected
ELSIF  i_stInfoData.usiMapDiag.4 = TRUE THEN
	q_sDiag := 'FSoE Slave Error Detected' ;

// Value		Description
// 0010 xxxx	FSoE Slave Reports Failsafe Value Active
ELSIF  i_stInfoData.usiMapDiag.5 = TRUE THEN
	q_sDiag := 'FSoE Slave Reports Failsafe Value Active' ;

// Value		Description
// 0100 xxxx	Connection is in Startup
ELSIF  i_stInfoData.usiMapDiag.6 = TRUE THEN
	q_sDiag := 'Connection Is In Startup' ;

// Value		Description
// 1000 xxxx	FSoE Master Reports Failsafe Value Active	
ELSIF  i_stInfoData.usiMapDiag.7 = TRUE THEN
	q_sDiag := 'FSoE Master Reports Failsafe Value Active' ;	

// Value		Description
//				Unknown Error
 				(* Something Not Specifically Annunciated Above.
 					possibly a combination OF errors are occuring. *)
ELSE	
	q_sDiag := 'Error' ;

END_IF

// Input Signals of the EP1908.
q_xSafIn1 := i_stInfoData.bInputSignals.0 ;
q_xSafIn2 := i_stInfoData.bInputSignals.1 ;
q_xSafIn3 := i_stInfoData.bInputSignals.2 ;
q_xSafIn4 := i_stInfoData.bInputSignals.3 ;
q_xSafIn5 := i_stInfoData.bInputSignals.4 ;
q_xSafIn6 := i_stInfoData.bInputSignals.5 ;
q_xSafIn7 := i_stInfoData.bInputSignals.6 ;
q_xSafIn8 := i_stInfoData.bInputSignals.7 ;

END_FUNCTION_BLOCK

// POUs/ConnectionAndFb_Blocks/Project/FB_SafetyConnectionGroup
(*=====================================================================
Beckhoff Automation LLC
Copyright 2015 All Rights Reserved
=======================================================================
Description: 
This Program has been supplied by Beckhoff Automation As-Is and is intended only as an example implementation. 
Functionality is not guaranteed. 
This Function Block reads status and error information known at time of creation of the TwinSAFE 'safery group'.
---------------------------------------------------------------------------------------------------------------
History:
Date		Version			Author							Comment
---------------------------------------------------------------------------------------------------------------
07.08.15	0.10		Jason Erickson				Initial Library Creation.
07.20.15	0.11		Jason Ericskon				Added CoE Read for TwinSAFE Connection State.
08.28.15	0.20		Jason Erickson				Code optimization to eliminate timed data reads.
09.18.15	0.2.1		Jason Erickson				Added new error codes 0x6000 - 0x6002 and Connection Status
														to the AX5805.
*)
FUNCTION_BLOCK FB_SafetyConnectionGroup
VAR_INPUT
(* ***** Structure linked to the 'TwinSAFE Group Info Data' of the EL69xx. ***** *)
	i_stInfoData: ST_SAFETY_CONNECTION_GROUP;
END_VAR
VAR_OUTPUT
// State of the EL2904 TwinSAFE Group.
	q_sState: STRING;
END_VAR

// Evaluate state of the TwinSAFE Group.

// Value 1 - RUN 
	(* All function blocks and TwinSAFE connections assigned to the TwinSAFE group operate properly, 
		and all TwinSAFE connections assigned to the TwinSAFE group are up and running. *)
IF i_stInfoData.usiMapState = 1 THEN
	q_sState := 'RUN - All FBs and Connections Operating Properly' ;

// Value 2 - Stop
	(* The state TwinSAFE goes to after initialization. *)
ELSIF i_stInfoData.usiMapState = 2 THEN
	q_sState := 'STOP - State After Initialization' ;

// Value 3 - SAFE 
	(* All function blocks and TwinSAFE connections assigned to the TwinSAFE group operate properly, 
		AND AT least one OF the TwinSAFE connections assigned TO the TwinSAFE group is NOT up AND running. *)
ELSIF i_stInfoData.usiMapState 	= 	3 THEN
	q_sState := 'SAFE - An Assigned Connection Not Up and Running' ;

// Value 4 - ERROR
	(* At least one assigned function block or one assigned TwinSAFE connection has reported an error. *)
	ELSIF i_stInfoData.usiMapState = 4 THEN
		q_sState := 'ERROR - FB or Connection in Error State' ;

// Value 5 - RESET
	(* A positive edge (FALSE -> TRUE) for the safety group error Ack of a function block or a TwinSAFE connection
		error was detected on the ERR_ACK input. The system is waiting for a negative edge of the ERR_ACK input. *)
ELSIF i_stInfoData.usiMapState = 5 THEN
	q_sState := 'RESET - ErrAck TRUE, Waiting For ErrAck FALSE' ;

// Safety group does not exist or safety controller has not been started.
ELSE
	q_sState := 'Unknown' ;
END_IF

// THE safery group HAS NO DIAGNOTIC BYTE TO DECODE!

END_FUNCTION_BLOCK

// POUs/HardwareFBs/FB_AX5805Diagnostics
(*=====================================================================
Beckhoff Automation LLC
Copyright 2015 All Rights Reserved
=======================================================================
Description: 
This Program has been supplied by Beckhoff Automation As-Is and is intended only as an example implementation. 
Functionality is not guaranteed. 
This Function Block reads all status and error information known at time of creation of the AX5805.
---------------------------------------------------------------------------------------------------------------
History:
Date		Version			Author							Comment
---------------------------------------------------------------------------------------------------------------
07.08.15	0.10		Jason Erickson				Initial Library Creation.
07.20.15	0.11		Jason Ericskon				Added CoE Read for TwinSAFE Connection State.
08.28.15	0.20		Jason Erickson				Code optimization to eliminate timed data reads.
09.18.15	0.2.1		Jason Erickson				Added new error codes 0x6000 - 0x6002 and Connection Status to the AX5805.
09.24.15	0.2.2		Jason Erickson				Corrected inability to update CASE in FB_EL1904Diagnostics and FB_EL2904Diagnostics.
10.30.15	0.2.3		Jason Erickson				Modified Diagnostic Structure names for ease of use.
*)
FUNCTION_BLOCK FB_AX5805Diagnostics
VAR_INPUT
	i_nSlaveAddr: UINT;		// Slave Address of the AX5805.
	i_nChooseChannel: UINT;	// Insert a 1 or a 2 to choose which AX5805 channel to read.
END_VAR
VAR_IN_OUT
	iq_stAxisRef: AXIS_REF;	// Axis Reference structure of the AX5000 Drive.
END_VAR
VAR_OUTPUT
	q_stAX5805_Diag: ST_AX5805_DIAGNOSTICS;	// Structure to hold all AX5805 output information.
	q_xError: BOOL;							// Function block Error.
	q_udiErrorID: UDINT;					// Function block Error ID.
	q_sErrorDescription: STRING;			// Function block Error Description.
END_VAR
VAR
//CASE Statement.
	iState: INT;
// FB_EcCoESdoRead for all CoE reads.
	fbCoERead: FB_EcCoESdoRead;
// FB and Structure to read/hold AX5000 Address Info.
	fbAX5000_ReadAddress: MC_ReadDriveAddress;
	stAX5000_DriveAddress: ST_DriveAddress;
// Variable to hold data for evaluation, Micro Controller (MC1) 3.3v Nominal Voltage(mV) INPUT of the AX5805.
	wAX5805_MC1_3300mV: WORD;
// Variable to hold data for evaluation, Micro Controller (MC1) 5.0v Nominal Voltage(mV) OUTPUT of the AX5805.
	wAX5805_MC1_5000mV: WORD;
// Variable to hold data for evaluation, Micro Controller (MC2) 3.3v Nominal Voltage(mV) INPUT of the AX5805.
	wAX5805_MC2_3300mV: WORD;
// Variable to hold data for evaluation, Micro Controller (MC2) 5.0v Nominal Voltage(mV) OUTPUT of the AX5805.
	wAX5805_MC2_5000mV: WORD;
// Variable to hold data for evaluation, Connection State of the AX5805.		
	iAX5805_ConnectionState: INT;
// Variable to hold data for evaluation, Configured Safety Option of the AX5000 Drive.
	fbAX5000_SafetyOptionSoeRead: FB_SoERead;
	wSafetyOption: WORD;
END_VAR

CASE iState OF
	0:// Read AX5000 EtherCAT Address Info.					
		fbAX5000_ReadAddress(
			Axis		  :=  iq_stAxisRef, 
			Execute		  :=  TRUE, 
			Done		  =>  , 
			Busy		  =>  , 
			Error		  =>  , 
			ErrorID		  =>  , 
			DriveAddress  =>  stAX5000_DriveAddress);

			iState := iState + 10;
			
	10:// Evaluate AX5000 EtherCAT Address Info.			
		fbAX5000_ReadAddress(Axis := iq_stAxisRef, Execute := TRUE); //Keep Alive.
		
		IF NOT fbAX5000_ReadAddress.Busy THEN
			fbAX5000_ReadAddress(Axis := iq_stAxisRef, Execute := FALSE);
			IF fbAX5000_ReadAddress.Error THEN
			q_udiErrorID := fbAX5000_ReadAddress.ErrorID;
				q_sErrorDescription := 'AX5000 EtherCAT Address - Read Error';
			ELSE
			q_sErrorDescription := 'No Error';
			END_IF
			iState := iState + 10;
		END_IF
	
	20:// Set Parameters to read the Serial Number of the AX5805.			
			fbCoERead.nSubIndex	:= 	16#02;
			fbCoERead.nIndex	:= 	16#F980;
			fbCoERead.pDstBuf	:= 	ADR(q_stAX5805_Diag.dwSerialNumber);
			fbCoERead.cbBufLen	:= 	SIZEOF(q_stAX5805_Diag.dwSerialNumber);
			fbCoERead.bExecute	:= 	TRUE;		
			iState := iState + 10;	
		
	30:// Evaluate read of the Serial Number of the AX5805.			
		IF NOT fbCoERead.bBusy THEN
			fbCoERead.bExecute := FALSE;
			q_sErrorDescription := 'No Error';
			iState := iState + 10;
			IF fbCoERead.bError THEN
				q_sErrorDescription := 'AX5805 Serial Number - Read Error';
			END_IF
		END_IF

	40:// Set Parameters to read the DIP Switch Setting of the AX5805.		
			fbCoERead.nSubIndex	:= 	16#01;
			fbCoERead.nIndex	:= 	16#F980;
			fbCoERead.pDstBuf	:= 	ADR(q_stAX5805_Diag.wDipSwitch);
			fbCoERead.cbBufLen	:= 	SIZEOF(q_stAX5805_Diag.wDipSwitch);
			fbCoERead.bExecute	:= 	TRUE;
			iState := iState + 10;	
			
	50:// Evaluate read of the DIP Switch Setting of the AX5805.		
		IF NOT fbCoERead.bBusy THEN
			fbCoERead.bExecute := FALSE;
			q_sErrorDescription := 'No Error';
			iState := iState + 10;
			IF fbCoERead.bError THEN
				q_sErrorDescription := 'AX5805 DIP Switch - Read Error';
			END_IF
		END_IF

	60:// Set Parameters to read the Hardware Version of the AX5805.		
			fbCoERead.nSubIndex	:= 	0;
			fbCoERead.nIndex	:= 	16#1009;
			fbCoERead.pDstBuf	:= 	ADR(q_stAX5805_Diag.sHwVersion);
			fbCoERead.cbBufLen	:= 	SIZEOF(q_stAX5805_Diag.sHwVersion);
			fbCoERead.bExecute	:= 	TRUE;
			iState := iState + 10;	
			
	70:// Evaluate read of the Hardware Version of the AX5805.		
		IF NOT fbCoERead.bBusy THEN
			fbCoERead.bExecute := FALSE;
			q_sErrorDescription := 'No Error';
			iState := iState + 10;
			IF fbCoERead.bError THEN
				q_sErrorDescription := 'AX5805 Hardware Version - Read Error';
			END_IF
		END_IF

	80:// Set Parameters to read the Software Version (firmware) of the AX5805.		
			fbCoERead.nSubIndex	:= 	0;
			fbCoERead.nIndex	:= 	16#100A;
			fbCoERead.pDstBuf	:= 	ADR(q_stAX5805_Diag.sFwVersion);
			fbCoERead.cbBufLen	:= 	SIZEOF(q_stAX5805_Diag.sFwVersion);
			fbCoERead.bExecute	:= 	TRUE;
			iState := iState + 10;	
			
	90:// Evaluate the Software Version (firmware) of the AX5805.		
		IF NOT fbCoERead.bBusy THEN
			fbCoERead.bExecute := FALSE;
			q_sErrorDescription := 'No Error';
			iState := iState + 10;
			IF fbCoERead.bError THEN
				q_sErrorDescription := 'AX5805 Software Version - Read Error';
			END_IF
		END_IF
		
	100:// Set Parameters to read the Micro Controller (MC1) Temperature in DegC of the AX5805.		
			fbCoERead.nSubIndex	:= 	16#01;
			fbCoERead.nIndex	:= 	16#FA80;
			fbCoERead.pDstBuf	:= 	ADR(q_stAX5805_Diag.wMC1Temp);
			fbCoERead.cbBufLen	:= 	SIZEOF(q_stAX5805_Diag.wMC1Temp);
			fbCoERead.bExecute	:= 	TRUE;
			iState := iState + 10;	
			
	110:// Evaluate the Micro Controller (MC1) Temperature in DegC of the AX5805.		
		IF NOT fbCoERead.bBusy THEN
			fbCoERead.bExecute := FALSE;
			q_sErrorDescription := 'No Error';
			iState := iState + 10;
			IF fbCoERead.bError THEN
				q_sErrorDescription := 'AX5805 MC1 Temp - Read Error';
			END_IF
		END_IF
		
	120:// Set Parameters to read the Micro Controller (MC2) Temperature in DegC of the AX5805.		
			fbCoERead.nSubIndex	:= 	16#02;
			fbCoERead.nIndex	:= 	16#FA80;
			fbCoERead.pDstBuf	:= 	ADR(q_stAX5805_Diag.wMC2Temp);
			fbCoERead.cbBufLen	:= 	SIZEOF(q_stAX5805_Diag.wMC2Temp);
			fbCoERead.bExecute	:= 	TRUE;
			iState := iState + 10;	
			
	130:// Evaluate the Micro Controller (MC2) Temperature in DegC of the AX5805.		
		IF NOT fbCoERead.bBusy THEN
			fbCoERead.bExecute := FALSE;
			q_sErrorDescription := 'No Error';
			iState := iState + 10;
			IF fbCoERead.bError THEN
				q_sErrorDescription := 'AX5805 MC2 Temp - Read Error';
			END_IF
		END_IF
	
	140:// Set Parameters to read the Micro Controller (MC1) 3300mv Nominal Voltage INPUT TO the AX5805.		
			fbCoERead.nSubIndex	:= 	16#01;
			fbCoERead.nIndex	:= 	16#FA81;
			fbCoERead.pDstBuf	:= 	ADR(wAX5805_MC1_3300mV);
			fbCoERead.cbBufLen	:= 	SIZEOF(wAX5805_MC1_3300mV);
			fbCoERead.bExecute	:= 	TRUE;
			iState := iState + 10;	
			
	150:// Evaluate the Micro Controller (MC1) 3300mv Nominal Voltage INPUT TO the AX5805.	
		IF NOT fbCoERead.bBusy THEN
			q_stAX5805_Diag.lrMC1_3300mV	:=  WORD_TO_LREAL(wAX5805_MC1_3300mV);
			fbCoERead.bExecute := FALSE;
			q_sErrorDescription := 'No Error';
			iState := iState + 10;
			IF fbCoERead.bError THEN
				q_sErrorDescription := 'AX5805 MC1 3.3v Input - Read Error';
			END_IF
		END_IF

	160:// Set Parameters to read the Micro Controller (MC1) 5000mv Nominal Voltage OUTPUT of the AX5805.		
			fbCoERead.nSubIndex	:= 	16#03;
			fbCoERead.nIndex	:= 	16#FA81;
			fbCoERead.pDstBuf	:= 	ADR(wAX5805_MC1_5000mV);
			fbCoERead.cbBufLen	:= 	SIZEOF(wAX5805_MC1_5000mV);
			fbCoERead.bExecute	:= 	TRUE;
			iState := iState + 10;	
			
	170:// Evaluate the Micro Controller (MC1) 5000mv Nominal Voltage OUTPUT of the AX5805.	
		IF NOT fbCoERead.bBusy THEN
			q_stAX5805_Diag.lrMC1_5000mV  :=  WORD_TO_LREAL(wAX5805_MC1_5000mV);
			fbCoERead.bExecute := FALSE;
			q_sErrorDescription := 'No Error';
			iState := iState + 10;
			IF fbCoERead.bError THEN
				q_sErrorDescription := 'AX5805 MC1 5.0v Output - Read Error';
			END_IF
		END_IF
		
	180:// Set Parameters to read the Micro Controller (MC2) 3.3v Nominal Voltage(mV) INPUT TO the AX5805.		
			fbCoERead.nSubIndex	:= 	16#02;
			fbCoERead.nIndex	:= 	16#FA81;
			fbCoERead.pDstBuf	:= 	ADR(wAX5805_MC2_3300mV);
			fbCoERead.cbBufLen	:= 	SIZEOF(wAX5805_MC2_3300mV);
			fbCoERead.bExecute	:= 	TRUE;
			iState := iState + 10;	
			
	190:// Evaluate the Micro Controller (MC2) 3.3v Nominal Voltage(mV) INPUT TO the AX5805.	
		IF NOT fbCoERead.bBusy THEN
		q_stAX5805_Diag.lrMC2_3300mV  :=  WORD_TO_LREAL(wAX5805_MC2_3300mV);
			fbCoERead.bExecute := FALSE;
			q_sErrorDescription := 'No Error';
			iState := iState + 10;
			IF fbCoERead.bError THEN
				q_sErrorDescription := 'AX5805 MC2 3.3v Input - Read Error';
			END_IF
		END_IF

	200:// Set Parameters to read the Micro Controller (MC2) 5.0v Nominal Voltage(mV) OUTPUT of the AX5805.		
			fbCoERead.nSubIndex	:= 	16#04;
			fbCoERead.nIndex	:= 	16#FA81;
			fbCoERead.pDstBuf	:= 	ADR(wAX5805_MC2_5000mV);
			fbCoERead.cbBufLen	:= 	SIZEOF(wAX5805_MC2_5000mV);
			fbCoERead.bExecute	:= 	TRUE;
			iState := iState + 10;	
			
	210:// Evaluate the Micro Controller (MC2) 5.0v Nominal Voltage(mV) OUTPUT of the AX5805.	
		IF NOT fbCoERead.bBusy THEN
		q_stAX5805_Diag.lrMC2_5000mV  :=  WORD_TO_LREAL(wAX5805_MC2_5000mV);
			fbCoERead.bExecute := FALSE;
			q_sErrorDescription := 'No Error';
			iState := iState + 10;
			IF fbCoERead.bError THEN
				q_sErrorDescription := 'AX5805 MC2 5.0v Output - Read Error';
			END_IF
		END_IF


